   // UNICODE_TO_GBK[22326] := 16#76CE;
   // UNICODE_TO_GBK[22327] := 16#B0BB;
   // UNICODE_TO_GBK[22328] := 16#76CF;
   // UNICODE_TO_GBK[22329] := 16#D5B5;
   // UNICODE_TO_GBK[22330] := 16#76D0;
   // UNICODE_TO_GBK[22331] := 16#D1CE;
   // UNICODE_TO_GBK[22332] := 16#76D1;
   // UNICODE_TO_GBK[22333] := 16#BCE0;
   // UNICODE_TO_GBK[22334] := 16#76D2;
   // UNICODE_TO_GBK[22335] := 16#BAD0;
   // UNICODE_TO_GBK[22336] := 16#76D3;
   // UNICODE_TO_GBK[22337] := 16#B145;
   // UNICODE_TO_GBK[22338] := 16#76D4;
   // UNICODE_TO_GBK[22339] := 16#BFF8;
   // UNICODE_TO_GBK[22340] := 16#76D5;
   // UNICODE_TO_GBK[22341] := 16#B146;
   // UNICODE_TO_GBK[22342] := 16#76D6;
   // UNICODE_TO_GBK[22343] := 16#B8C7;
   // UNICODE_TO_GBK[22344] := 16#76D7;
   // UNICODE_TO_GBK[22345] := 16#B5C1;
   // UNICODE_TO_GBK[22346] := 16#76D8;
   // UNICODE_TO_GBK[22347] := 16#C5CC;
   // UNICODE_TO_GBK[22348] := 16#76D9;
   // UNICODE_TO_GBK[22349] := 16#B147;
   // UNICODE_TO_GBK[22350] := 16#76DA;
   // UNICODE_TO_GBK[22351] := 16#B148;
   // UNICODE_TO_GBK[22352] := 16#76DB;
   // UNICODE_TO_GBK[22353] := 16#CAA2;
   // UNICODE_TO_GBK[22354] := 16#76DC;
   // UNICODE_TO_GBK[22355] := 16#B149;
   // UNICODE_TO_GBK[22356] := 16#76DD;
   // UNICODE_TO_GBK[22357] := 16#B14A;
   // UNICODE_TO_GBK[22358] := 16#76DE;
   // UNICODE_TO_GBK[22359] := 16#B14B;
   // UNICODE_TO_GBK[22360] := 16#76DF;
   // UNICODE_TO_GBK[22361] := 16#C3CB;
   // UNICODE_TO_GBK[22362] := 16#76E0;
   // UNICODE_TO_GBK[22363] := 16#B14C;
   // UNICODE_TO_GBK[22364] := 16#76E1;
   // UNICODE_TO_GBK[22365] := 16#B14D;
   // UNICODE_TO_GBK[22366] := 16#76E2;
   // UNICODE_TO_GBK[22367] := 16#B14E;
   // UNICODE_TO_GBK[22368] := 16#76E3;
   // UNICODE_TO_GBK[22369] := 16#B14F;
   // UNICODE_TO_GBK[22370] := 16#76E4;
   // UNICODE_TO_GBK[22371] := 16#B150;
   // UNICODE_TO_GBK[22372] := 16#76E5;
   // UNICODE_TO_GBK[22373] := 16#EEC2;
   // UNICODE_TO_GBK[22374] := 16#76E6;
   // UNICODE_TO_GBK[22375] := 16#B151;
   // UNICODE_TO_GBK[22376] := 16#76E7;
   // UNICODE_TO_GBK[22377] := 16#B152;
   // UNICODE_TO_GBK[22378] := 16#76E8;
   // UNICODE_TO_GBK[22379] := 16#B153;
   // UNICODE_TO_GBK[22380] := 16#76E9;
   // UNICODE_TO_GBK[22381] := 16#B154;
   // UNICODE_TO_GBK[22382] := 16#76EA;
   // UNICODE_TO_GBK[22383] := 16#B155;
   // UNICODE_TO_GBK[22384] := 16#76EB;
   // UNICODE_TO_GBK[22385] := 16#B156;
   // UNICODE_TO_GBK[22386] := 16#76EC;
   // UNICODE_TO_GBK[22387] := 16#B157;
   // UNICODE_TO_GBK[22388] := 16#76ED;
   // UNICODE_TO_GBK[22389] := 16#B158;
   // UNICODE_TO_GBK[22390] := 16#76EE;
   // UNICODE_TO_GBK[22391] := 16#C4BF;
   // UNICODE_TO_GBK[22392] := 16#76EF;
   // UNICODE_TO_GBK[22393] := 16#B6A2;
   // UNICODE_TO_GBK[22394] := 16#76F0;
   // UNICODE_TO_GBK[22395] := 16#B159;
   // UNICODE_TO_GBK[22396] := 16#76F1;
   // UNICODE_TO_GBK[22397] := 16#EDEC;
   // UNICODE_TO_GBK[22398] := 16#76F2;
   // UNICODE_TO_GBK[22399] := 16#C3A4;
   // UNICODE_TO_GBK[22400] := 16#76F3;
   // UNICODE_TO_GBK[22401] := 16#B15A;
   // UNICODE_TO_GBK[22402] := 16#76F4;
   // UNICODE_TO_GBK[22403] := 16#D6B1;
   // UNICODE_TO_GBK[22404] := 16#76F5;
   // UNICODE_TO_GBK[22405] := 16#B15B;
   // UNICODE_TO_GBK[22406] := 16#76F6;
   // UNICODE_TO_GBK[22407] := 16#B15C;
   // UNICODE_TO_GBK[22408] := 16#76F7;
   // UNICODE_TO_GBK[22409] := 16#B15D;
   // UNICODE_TO_GBK[22410] := 16#76F8;
   // UNICODE_TO_GBK[22411] := 16#CFE0;
   // UNICODE_TO_GBK[22412] := 16#76F9;
   // UNICODE_TO_GBK[22413] := 16#EDEF;
   // UNICODE_TO_GBK[22414] := 16#76FA;
   // UNICODE_TO_GBK[22415] := 16#B15E;
   // UNICODE_TO_GBK[22416] := 16#76FB;
   // UNICODE_TO_GBK[22417] := 16#B15F;
   // UNICODE_TO_GBK[22418] := 16#76FC;
   // UNICODE_TO_GBK[22419] := 16#C5CE;
   // UNICODE_TO_GBK[22420] := 16#76FD;
   // UNICODE_TO_GBK[22421] := 16#B160;
   // UNICODE_TO_GBK[22422] := 16#76FE;
   // UNICODE_TO_GBK[22423] := 16#B6DC;
   // UNICODE_TO_GBK[22424] := 16#76FF;
   // UNICODE_TO_GBK[22425] := 16#B161;
   // UNICODE_TO_GBK[22426] := 16#7700;
   // UNICODE_TO_GBK[22427] := 16#B162;
   // UNICODE_TO_GBK[22428] := 16#7701;
   // UNICODE_TO_GBK[22429] := 16#CAA1;
   // UNICODE_TO_GBK[22430] := 16#7702;
   // UNICODE_TO_GBK[22431] := 16#B163;
   // UNICODE_TO_GBK[22432] := 16#7703;
   // UNICODE_TO_GBK[22433] := 16#B164;
   // UNICODE_TO_GBK[22434] := 16#7704;
   // UNICODE_TO_GBK[22435] := 16#EDED;
   // UNICODE_TO_GBK[22436] := 16#7705;
   // UNICODE_TO_GBK[22437] := 16#B165;
   // UNICODE_TO_GBK[22438] := 16#7706;
   // UNICODE_TO_GBK[22439] := 16#B166;
   // UNICODE_TO_GBK[22440] := 16#7707;
   // UNICODE_TO_GBK[22441] := 16#EDF0;
   // UNICODE_TO_GBK[22442] := 16#7708;
   // UNICODE_TO_GBK[22443] := 16#EDF1;
   // UNICODE_TO_GBK[22444] := 16#7709;
   // UNICODE_TO_GBK[22445] := 16#C3BC;
   // UNICODE_TO_GBK[22446] := 16#770A;
   // UNICODE_TO_GBK[22447] := 16#B167;
   // UNICODE_TO_GBK[22448] := 16#770B;
   // UNICODE_TO_GBK[22449] := 16#BFB4;
   // UNICODE_TO_GBK[22450] := 16#770C;
   // UNICODE_TO_GBK[22451] := 16#B168;
   // UNICODE_TO_GBK[22452] := 16#770D;
   // UNICODE_TO_GBK[22453] := 16#EDEE;
   // UNICODE_TO_GBK[22454] := 16#770E;
   // UNICODE_TO_GBK[22455] := 16#B169;
   // UNICODE_TO_GBK[22456] := 16#770F;
   // UNICODE_TO_GBK[22457] := 16#B16A;
   // UNICODE_TO_GBK[22458] := 16#7710;
   // UNICODE_TO_GBK[22459] := 16#B16B;
   // UNICODE_TO_GBK[22460] := 16#7711;
   // UNICODE_TO_GBK[22461] := 16#B16C;
   // UNICODE_TO_GBK[22462] := 16#7712;
   // UNICODE_TO_GBK[22463] := 16#B16D;
   // UNICODE_TO_GBK[22464] := 16#7713;
   // UNICODE_TO_GBK[22465] := 16#B16E;
   // UNICODE_TO_GBK[22466] := 16#7714;
   // UNICODE_TO_GBK[22467] := 16#B16F;
   // UNICODE_TO_GBK[22468] := 16#7715;
   // UNICODE_TO_GBK[22469] := 16#B170;
   // UNICODE_TO_GBK[22470] := 16#7716;
   // UNICODE_TO_GBK[22471] := 16#B171;
   // UNICODE_TO_GBK[22472] := 16#7717;
   // UNICODE_TO_GBK[22473] := 16#B172;
   // UNICODE_TO_GBK[22474] := 16#7718;
   // UNICODE_TO_GBK[22475] := 16#B173;
   // UNICODE_TO_GBK[22476] := 16#7719;
   // UNICODE_TO_GBK[22477] := 16#EDF4;
   // UNICODE_TO_GBK[22478] := 16#771A;
   // UNICODE_TO_GBK[22479] := 16#EDF2;
   // UNICODE_TO_GBK[22480] := 16#771B;
   // UNICODE_TO_GBK[22481] := 16#B174;
   // UNICODE_TO_GBK[22482] := 16#771C;
   // UNICODE_TO_GBK[22483] := 16#B175;
   // UNICODE_TO_GBK[22484] := 16#771D;
   // UNICODE_TO_GBK[22485] := 16#B176;
   // UNICODE_TO_GBK[22486] := 16#771E;
   // UNICODE_TO_GBK[22487] := 16#B177;
   // UNICODE_TO_GBK[22488] := 16#771F;
   // UNICODE_TO_GBK[22489] := 16#D5E6;
   // UNICODE_TO_GBK[22490] := 16#7720;
   // UNICODE_TO_GBK[22491] := 16#C3DF;
   // UNICODE_TO_GBK[22492] := 16#7721;
   // UNICODE_TO_GBK[22493] := 16#B178;
   // UNICODE_TO_GBK[22494] := 16#7722;
   // UNICODE_TO_GBK[22495] := 16#EDF3;
   // UNICODE_TO_GBK[22496] := 16#7723;
   // UNICODE_TO_GBK[22497] := 16#B179;
   // UNICODE_TO_GBK[22498] := 16#7724;
   // UNICODE_TO_GBK[22499] := 16#B17A;
   // UNICODE_TO_GBK[22500] := 16#7725;
   // UNICODE_TO_GBK[22501] := 16#B17B;
   // UNICODE_TO_GBK[22502] := 16#7726;
   // UNICODE_TO_GBK[22503] := 16#EDF6;
   // UNICODE_TO_GBK[22504] := 16#7727;
   // UNICODE_TO_GBK[22505] := 16#B17C;
   // UNICODE_TO_GBK[22506] := 16#7728;
   // UNICODE_TO_GBK[22507] := 16#D5A3;
   // UNICODE_TO_GBK[22508] := 16#7729;
   // UNICODE_TO_GBK[22509] := 16#D1A3;
   // UNICODE_TO_GBK[22510] := 16#772A;
   // UNICODE_TO_GBK[22511] := 16#B17D;
   // UNICODE_TO_GBK[22512] := 16#772B;
   // UNICODE_TO_GBK[22513] := 16#B17E;
   // UNICODE_TO_GBK[22514] := 16#772C;
   // UNICODE_TO_GBK[22515] := 16#B180;
   // UNICODE_TO_GBK[22516] := 16#772D;
   // UNICODE_TO_GBK[22517] := 16#EDF5;
   // UNICODE_TO_GBK[22518] := 16#772E;
   // UNICODE_TO_GBK[22519] := 16#B181;
   // UNICODE_TO_GBK[22520] := 16#772F;
   // UNICODE_TO_GBK[22521] := 16#C3D0;
   // UNICODE_TO_GBK[22522] := 16#7730;
   // UNICODE_TO_GBK[22523] := 16#B182;
   // UNICODE_TO_GBK[22524] := 16#7731;
   // UNICODE_TO_GBK[22525] := 16#B183;
   // UNICODE_TO_GBK[22526] := 16#7732;
   // UNICODE_TO_GBK[22527] := 16#B184;
   // UNICODE_TO_GBK[22528] := 16#7733;
   // UNICODE_TO_GBK[22529] := 16#B185;
   // UNICODE_TO_GBK[22530] := 16#7734;
   // UNICODE_TO_GBK[22531] := 16#B186;
   // UNICODE_TO_GBK[22532] := 16#7735;
   // UNICODE_TO_GBK[22533] := 16#EDF7;
   // UNICODE_TO_GBK[22534] := 16#7736;
   // UNICODE_TO_GBK[22535] := 16#BFF4;
   // UNICODE_TO_GBK[22536] := 16#7737;
   // UNICODE_TO_GBK[22537] := 16#BEEC;
   // UNICODE_TO_GBK[22538] := 16#7738;
   // UNICODE_TO_GBK[22539] := 16#EDF8;
   // UNICODE_TO_GBK[22540] := 16#7739;
   // UNICODE_TO_GBK[22541] := 16#B187;
   // UNICODE_TO_GBK[22542] := 16#773A;
   // UNICODE_TO_GBK[22543] := 16#CCF7;
   // UNICODE_TO_GBK[22544] := 16#773B;
   // UNICODE_TO_GBK[22545] := 16#B188;
   // UNICODE_TO_GBK[22546] := 16#773C;
   // UNICODE_TO_GBK[22547] := 16#D1DB;
   // UNICODE_TO_GBK[22548] := 16#773D;
   // UNICODE_TO_GBK[22549] := 16#B189;
   // UNICODE_TO_GBK[22550] := 16#773E;
   // UNICODE_TO_GBK[22551] := 16#B18A;
   // UNICODE_TO_GBK[22552] := 16#773F;
   // UNICODE_TO_GBK[22553] := 16#B18B;
   // UNICODE_TO_GBK[22554] := 16#7740;
   // UNICODE_TO_GBK[22555] := 16#D7C5;
   // UNICODE_TO_GBK[22556] := 16#7741;
   // UNICODE_TO_GBK[22557] := 16#D5F6;
   // UNICODE_TO_GBK[22558] := 16#7742;
   // UNICODE_TO_GBK[22559] := 16#B18C;
   // UNICODE_TO_GBK[22560] := 16#7743;
   // UNICODE_TO_GBK[22561] := 16#EDFC;
   // UNICODE_TO_GBK[22562] := 16#7744;
   // UNICODE_TO_GBK[22563] := 16#B18D;
   // UNICODE_TO_GBK[22564] := 16#7745;
   // UNICODE_TO_GBK[22565] := 16#B18E;
   // UNICODE_TO_GBK[22566] := 16#7746;
   // UNICODE_TO_GBK[22567] := 16#B18F;
   // UNICODE_TO_GBK[22568] := 16#7747;
   // UNICODE_TO_GBK[22569] := 16#EDFB;
   // UNICODE_TO_GBK[22570] := 16#7748;
   // UNICODE_TO_GBK[22571] := 16#B190;
   // UNICODE_TO_GBK[22572] := 16#7749;
   // UNICODE_TO_GBK[22573] := 16#B191;
   // UNICODE_TO_GBK[22574] := 16#774A;
   // UNICODE_TO_GBK[22575] := 16#B192;
   // UNICODE_TO_GBK[22576] := 16#774B;
   // UNICODE_TO_GBK[22577] := 16#B193;
   // UNICODE_TO_GBK[22578] := 16#774C;
   // UNICODE_TO_GBK[22579] := 16#B194;
   // UNICODE_TO_GBK[22580] := 16#774D;
   // UNICODE_TO_GBK[22581] := 16#B195;
   // UNICODE_TO_GBK[22582] := 16#774E;
   // UNICODE_TO_GBK[22583] := 16#B196;
   // UNICODE_TO_GBK[22584] := 16#774F;
   // UNICODE_TO_GBK[22585] := 16#B197;
   // UNICODE_TO_GBK[22586] := 16#7750;
   // UNICODE_TO_GBK[22587] := 16#EDF9;
   // UNICODE_TO_GBK[22588] := 16#7751;
   // UNICODE_TO_GBK[22589] := 16#EDFA;
   // UNICODE_TO_GBK[22590] := 16#7752;
   // UNICODE_TO_GBK[22591] := 16#B198;
   // UNICODE_TO_GBK[22592] := 16#7753;
   // UNICODE_TO_GBK[22593] := 16#B199;
   // UNICODE_TO_GBK[22594] := 16#7754;
   // UNICODE_TO_GBK[22595] := 16#B19A;
   // UNICODE_TO_GBK[22596] := 16#7755;
   // UNICODE_TO_GBK[22597] := 16#B19B;
   // UNICODE_TO_GBK[22598] := 16#7756;
   // UNICODE_TO_GBK[22599] := 16#B19C;
   // UNICODE_TO_GBK[22600] := 16#7757;
   // UNICODE_TO_GBK[22601] := 16#B19D;
   // UNICODE_TO_GBK[22602] := 16#7758;
   // UNICODE_TO_GBK[22603] := 16#B19E;
   // UNICODE_TO_GBK[22604] := 16#7759;
   // UNICODE_TO_GBK[22605] := 16#B19F;
   // UNICODE_TO_GBK[22606] := 16#775A;
   // UNICODE_TO_GBK[22607] := 16#EDFD;
   // UNICODE_TO_GBK[22608] := 16#775B;
   // UNICODE_TO_GBK[22609] := 16#BEA6;
   // UNICODE_TO_GBK[22610] := 16#775C;
   // UNICODE_TO_GBK[22611] := 16#B1A0;
   // UNICODE_TO_GBK[22612] := 16#775D;
   // UNICODE_TO_GBK[22613] := 16#B240;
   // UNICODE_TO_GBK[22614] := 16#775E;
   // UNICODE_TO_GBK[22615] := 16#B241;
   // UNICODE_TO_GBK[22616] := 16#775F;
   // UNICODE_TO_GBK[22617] := 16#B242;
   // UNICODE_TO_GBK[22618] := 16#7760;
   // UNICODE_TO_GBK[22619] := 16#B243;
   // UNICODE_TO_GBK[22620] := 16#7761;
   // UNICODE_TO_GBK[22621] := 16#CBAF;
   // UNICODE_TO_GBK[22622] := 16#7762;
   // UNICODE_TO_GBK[22623] := 16#EEA1;
   // UNICODE_TO_GBK[22624] := 16#7763;
   // UNICODE_TO_GBK[22625] := 16#B6BD;
   // UNICODE_TO_GBK[22626] := 16#7764;
   // UNICODE_TO_GBK[22627] := 16#B244;
   // UNICODE_TO_GBK[22628] := 16#7765;
   // UNICODE_TO_GBK[22629] := 16#EEA2;
   // UNICODE_TO_GBK[22630] := 16#7766;
   // UNICODE_TO_GBK[22631] := 16#C4C0;
   // UNICODE_TO_GBK[22632] := 16#7767;
   // UNICODE_TO_GBK[22633] := 16#B245;
   // UNICODE_TO_GBK[22634] := 16#7768;
   // UNICODE_TO_GBK[22635] := 16#EDFE;
   // UNICODE_TO_GBK[22636] := 16#7769;
   // UNICODE_TO_GBK[22637] := 16#B246;
   // UNICODE_TO_GBK[22638] := 16#776A;
   // UNICODE_TO_GBK[22639] := 16#B247;
   // UNICODE_TO_GBK[22640] := 16#776B;
   // UNICODE_TO_GBK[22641] := 16#BDDE;
   // UNICODE_TO_GBK[22642] := 16#776C;
   // UNICODE_TO_GBK[22643] := 16#B2C7;
   // UNICODE_TO_GBK[22644] := 16#776D;
   // UNICODE_TO_GBK[22645] := 16#B248;
   // UNICODE_TO_GBK[22646] := 16#776E;
   // UNICODE_TO_GBK[22647] := 16#B249;
   // UNICODE_TO_GBK[22648] := 16#776F;
   // UNICODE_TO_GBK[22649] := 16#B24A;
   // UNICODE_TO_GBK[22650] := 16#7770;
   // UNICODE_TO_GBK[22651] := 16#B24B;
   // UNICODE_TO_GBK[22652] := 16#7771;
   // UNICODE_TO_GBK[22653] := 16#B24C;
   // UNICODE_TO_GBK[22654] := 16#7772;
   // UNICODE_TO_GBK[22655] := 16#B24D;
   // UNICODE_TO_GBK[22656] := 16#7773;
   // UNICODE_TO_GBK[22657] := 16#B24E;
   // UNICODE_TO_GBK[22658] := 16#7774;
   // UNICODE_TO_GBK[22659] := 16#B24F;
   // UNICODE_TO_GBK[22660] := 16#7775;
   // UNICODE_TO_GBK[22661] := 16#B250;
   // UNICODE_TO_GBK[22662] := 16#7776;
   // UNICODE_TO_GBK[22663] := 16#B251;
   // UNICODE_TO_GBK[22664] := 16#7777;
   // UNICODE_TO_GBK[22665] := 16#B252;
   // UNICODE_TO_GBK[22666] := 16#7778;
   // UNICODE_TO_GBK[22667] := 16#B253;
   // UNICODE_TO_GBK[22668] := 16#7779;
   // UNICODE_TO_GBK[22669] := 16#B6C3;
   // UNICODE_TO_GBK[22670] := 16#777A;
   // UNICODE_TO_GBK[22671] := 16#B254;
   // UNICODE_TO_GBK[22672] := 16#777B;
   // UNICODE_TO_GBK[22673] := 16#B255;
   // UNICODE_TO_GBK[22674] := 16#777C;
   // UNICODE_TO_GBK[22675] := 16#B256;
   // UNICODE_TO_GBK[22676] := 16#777D;
   // UNICODE_TO_GBK[22677] := 16#EEA5;
   // UNICODE_TO_GBK[22678] := 16#777E;
   // UNICODE_TO_GBK[22679] := 16#D8BA;
   // UNICODE_TO_GBK[22680] := 16#777F;
   // UNICODE_TO_GBK[22681] := 16#EEA3;
   // UNICODE_TO_GBK[22682] := 16#7780;
   // UNICODE_TO_GBK[22683] := 16#EEA6;
   // UNICODE_TO_GBK[22684] := 16#7781;
   // UNICODE_TO_GBK[22685] := 16#B257;
   // UNICODE_TO_GBK[22686] := 16#7782;
   // UNICODE_TO_GBK[22687] := 16#B258;
   // UNICODE_TO_GBK[22688] := 16#7783;
   // UNICODE_TO_GBK[22689] := 16#B259;
   // UNICODE_TO_GBK[22690] := 16#7784;
   // UNICODE_TO_GBK[22691] := 16#C3E9;
   // UNICODE_TO_GBK[22692] := 16#7785;
   // UNICODE_TO_GBK[22693] := 16#B3F2;
   // UNICODE_TO_GBK[22694] := 16#7786;
   // UNICODE_TO_GBK[22695] := 16#B25A;
   // UNICODE_TO_GBK[22696] := 16#7787;
   // UNICODE_TO_GBK[22697] := 16#B25B;
   // UNICODE_TO_GBK[22698] := 16#7788;
   // UNICODE_TO_GBK[22699] := 16#B25C;
   // UNICODE_TO_GBK[22700] := 16#7789;
   // UNICODE_TO_GBK[22701] := 16#B25D;
   // UNICODE_TO_GBK[22702] := 16#778A;
   // UNICODE_TO_GBK[22703] := 16#B25E;
   // UNICODE_TO_GBK[22704] := 16#778B;
   // UNICODE_TO_GBK[22705] := 16#B25F;
   // UNICODE_TO_GBK[22706] := 16#778C;
   // UNICODE_TO_GBK[22707] := 16#EEA7;
   // UNICODE_TO_GBK[22708] := 16#778D;
   // UNICODE_TO_GBK[22709] := 16#EEA4;
   // UNICODE_TO_GBK[22710] := 16#778E;
   // UNICODE_TO_GBK[22711] := 16#CFB9;
   // UNICODE_TO_GBK[22712] := 16#778F;
   // UNICODE_TO_GBK[22713] := 16#B260;
   // UNICODE_TO_GBK[22714] := 16#7790;
   // UNICODE_TO_GBK[22715] := 16#B261;
   // UNICODE_TO_GBK[22716] := 16#7791;
   // UNICODE_TO_GBK[22717] := 16#EEA8;
   // UNICODE_TO_GBK[22718] := 16#7792;
   // UNICODE_TO_GBK[22719] := 16#C2F7;
   // UNICODE_TO_GBK[22720] := 16#7793;
   // UNICODE_TO_GBK[22721] := 16#B262;
   // UNICODE_TO_GBK[22722] := 16#7794;
   // UNICODE_TO_GBK[22723] := 16#B263;
   // UNICODE_TO_GBK[22724] := 16#7795;
   // UNICODE_TO_GBK[22725] := 16#B264;
   // UNICODE_TO_GBK[22726] := 16#7796;
   // UNICODE_TO_GBK[22727] := 16#B265;
   // UNICODE_TO_GBK[22728] := 16#7797;
   // UNICODE_TO_GBK[22729] := 16#B266;
   // UNICODE_TO_GBK[22730] := 16#7798;
   // UNICODE_TO_GBK[22731] := 16#B267;
   // UNICODE_TO_GBK[22732] := 16#7799;
   // UNICODE_TO_GBK[22733] := 16#B268;
   // UNICODE_TO_GBK[22734] := 16#779A;
   // UNICODE_TO_GBK[22735] := 16#B269;
   // UNICODE_TO_GBK[22736] := 16#779B;
   // UNICODE_TO_GBK[22737] := 16#B26A;
   // UNICODE_TO_GBK[22738] := 16#779C;
   // UNICODE_TO_GBK[22739] := 16#B26B;
   // UNICODE_TO_GBK[22740] := 16#779D;
   // UNICODE_TO_GBK[22741] := 16#B26C;
   // UNICODE_TO_GBK[22742] := 16#779E;
   // UNICODE_TO_GBK[22743] := 16#B26D;
   // UNICODE_TO_GBK[22744] := 16#779F;
   // UNICODE_TO_GBK[22745] := 16#EEA9;
   // UNICODE_TO_GBK[22746] := 16#77A0;
   // UNICODE_TO_GBK[22747] := 16#EEAA;
   // UNICODE_TO_GBK[22748] := 16#77A1;
   // UNICODE_TO_GBK[22749] := 16#B26E;
   // UNICODE_TO_GBK[22750] := 16#77A2;
   // UNICODE_TO_GBK[22751] := 16#DEAB;
   // UNICODE_TO_GBK[22752] := 16#77A3;
   // UNICODE_TO_GBK[22753] := 16#B26F;
   // UNICODE_TO_GBK[22754] := 16#77A4;
   // UNICODE_TO_GBK[22755] := 16#B270;
   // UNICODE_TO_GBK[22756] := 16#77A5;
   // UNICODE_TO_GBK[22757] := 16#C6B3;
   // UNICODE_TO_GBK[22758] := 16#77A6;
   // UNICODE_TO_GBK[22759] := 16#B271;
   // UNICODE_TO_GBK[22760] := 16#77A7;
   // UNICODE_TO_GBK[22761] := 16#C7C6;
   // UNICODE_TO_GBK[22762] := 16#77A8;
   // UNICODE_TO_GBK[22763] := 16#B272;
   // UNICODE_TO_GBK[22764] := 16#77A9;
   // UNICODE_TO_GBK[22765] := 16#D6F5;
   // UNICODE_TO_GBK[22766] := 16#77AA;
   // UNICODE_TO_GBK[22767] := 16#B5C9;
   // UNICODE_TO_GBK[22768] := 16#77AB;
   // UNICODE_TO_GBK[22769] := 16#B273;
   // UNICODE_TO_GBK[22770] := 16#77AC;
   // UNICODE_TO_GBK[22771] := 16#CBB2;
   // UNICODE_TO_GBK[22772] := 16#77AD;
   // UNICODE_TO_GBK[22773] := 16#B274;
   // UNICODE_TO_GBK[22774] := 16#77AE;
   // UNICODE_TO_GBK[22775] := 16#B275;
   // UNICODE_TO_GBK[22776] := 16#77AF;
   // UNICODE_TO_GBK[22777] := 16#B276;
   // UNICODE_TO_GBK[22778] := 16#77B0;
   // UNICODE_TO_GBK[22779] := 16#EEAB;
   // UNICODE_TO_GBK[22780] := 16#77B1;
   // UNICODE_TO_GBK[22781] := 16#B277;
   // UNICODE_TO_GBK[22782] := 16#77B2;
   // UNICODE_TO_GBK[22783] := 16#B278;
   // UNICODE_TO_GBK[22784] := 16#77B3;
   // UNICODE_TO_GBK[22785] := 16#CDAB;
   // UNICODE_TO_GBK[22786] := 16#77B4;
   // UNICODE_TO_GBK[22787] := 16#B279;
   // UNICODE_TO_GBK[22788] := 16#77B5;
   // UNICODE_TO_GBK[22789] := 16#EEAC;
   // UNICODE_TO_GBK[22790] := 16#77B6;
   // UNICODE_TO_GBK[22791] := 16#B27A;
   // UNICODE_TO_GBK[22792] := 16#77B7;
   // UNICODE_TO_GBK[22793] := 16#B27B;
   // UNICODE_TO_GBK[22794] := 16#77B8;
   // UNICODE_TO_GBK[22795] := 16#B27C;
   // UNICODE_TO_GBK[22796] := 16#77B9;
   // UNICODE_TO_GBK[22797] := 16#B27D;
   // UNICODE_TO_GBK[22798] := 16#77BA;
   // UNICODE_TO_GBK[22799] := 16#B27E;
   // UNICODE_TO_GBK[22800] := 16#77BB;
   // UNICODE_TO_GBK[22801] := 16#D5B0;
   // UNICODE_TO_GBK[22802] := 16#77BC;
   // UNICODE_TO_GBK[22803] := 16#B280;
   // UNICODE_TO_GBK[22804] := 16#77BD;
   // UNICODE_TO_GBK[22805] := 16#EEAD;
   // UNICODE_TO_GBK[22806] := 16#77BE;
   // UNICODE_TO_GBK[22807] := 16#B281;
   // UNICODE_TO_GBK[22808] := 16#77BF;
   // UNICODE_TO_GBK[22809] := 16#F6C4;
   // UNICODE_TO_GBK[22810] := 16#77C0;
   // UNICODE_TO_GBK[22811] := 16#B282;
   // UNICODE_TO_GBK[22812] := 16#77C1;
   // UNICODE_TO_GBK[22813] := 16#B283;
   // UNICODE_TO_GBK[22814] := 16#77C2;
   // UNICODE_TO_GBK[22815] := 16#B284;
   // UNICODE_TO_GBK[22816] := 16#77C3;
   // UNICODE_TO_GBK[22817] := 16#B285;
   // UNICODE_TO_GBK[22818] := 16#77C4;
   // UNICODE_TO_GBK[22819] := 16#B286;
   // UNICODE_TO_GBK[22820] := 16#77C5;
   // UNICODE_TO_GBK[22821] := 16#B287;
   // UNICODE_TO_GBK[22822] := 16#77C6;
   // UNICODE_TO_GBK[22823] := 16#B288;
   // UNICODE_TO_GBK[22824] := 16#77C7;
   // UNICODE_TO_GBK[22825] := 16#B289;
   // UNICODE_TO_GBK[22826] := 16#77C8;
   // UNICODE_TO_GBK[22827] := 16#B28A;
   // UNICODE_TO_GBK[22828] := 16#77C9;
   // UNICODE_TO_GBK[22829] := 16#B28B;
   // UNICODE_TO_GBK[22830] := 16#77CA;
   // UNICODE_TO_GBK[22831] := 16#B28C;
   // UNICODE_TO_GBK[22832] := 16#77CB;
   // UNICODE_TO_GBK[22833] := 16#B28D;
   // UNICODE_TO_GBK[22834] := 16#77CC;
   // UNICODE_TO_GBK[22835] := 16#B28E;
   // UNICODE_TO_GBK[22836] := 16#77CD;
   // UNICODE_TO_GBK[22837] := 16#DBC7;
   // UNICODE_TO_GBK[22838] := 16#77CE;
   // UNICODE_TO_GBK[22839] := 16#B28F;
   // UNICODE_TO_GBK[22840] := 16#77CF;
   // UNICODE_TO_GBK[22841] := 16#B290;
   // UNICODE_TO_GBK[22842] := 16#77D0;
   // UNICODE_TO_GBK[22843] := 16#B291;
   // UNICODE_TO_GBK[22844] := 16#77D1;
   // UNICODE_TO_GBK[22845] := 16#B292;
   // UNICODE_TO_GBK[22846] := 16#77D2;
   // UNICODE_TO_GBK[22847] := 16#B293;
   // UNICODE_TO_GBK[22848] := 16#77D3;
   // UNICODE_TO_GBK[22849] := 16#B294;
   // UNICODE_TO_GBK[22850] := 16#77D4;
   // UNICODE_TO_GBK[22851] := 16#B295;
   // UNICODE_TO_GBK[22852] := 16#77D5;
   // UNICODE_TO_GBK[22853] := 16#B296;
   // UNICODE_TO_GBK[22854] := 16#77D6;
   // UNICODE_TO_GBK[22855] := 16#B297;
   // UNICODE_TO_GBK[22856] := 16#77D7;
   // UNICODE_TO_GBK[22857] := 16#B4A3;
   // UNICODE_TO_GBK[22858] := 16#77D8;
   // UNICODE_TO_GBK[22859] := 16#B298;
   // UNICODE_TO_GBK[22860] := 16#77D9;
   // UNICODE_TO_GBK[22861] := 16#B299;
   // UNICODE_TO_GBK[22862] := 16#77DA;
   // UNICODE_TO_GBK[22863] := 16#B29A;
   // UNICODE_TO_GBK[22864] := 16#77DB;
   // UNICODE_TO_GBK[22865] := 16#C3AC;
   // UNICODE_TO_GBK[22866] := 16#77DC;
   // UNICODE_TO_GBK[22867] := 16#F1E6;
   // UNICODE_TO_GBK[22868] := 16#77DD;
   // UNICODE_TO_GBK[22869] := 16#B29B;
   // UNICODE_TO_GBK[22870] := 16#77DE;
   // UNICODE_TO_GBK[22871] := 16#B29C;
   // UNICODE_TO_GBK[22872] := 16#77DF;
   // UNICODE_TO_GBK[22873] := 16#B29D;
   // UNICODE_TO_GBK[22874] := 16#77E0;
   // UNICODE_TO_GBK[22875] := 16#B29E;
   // UNICODE_TO_GBK[22876] := 16#77E1;
   // UNICODE_TO_GBK[22877] := 16#B29F;
   // UNICODE_TO_GBK[22878] := 16#77E2;
   // UNICODE_TO_GBK[22879] := 16#CAB8;
   // UNICODE_TO_GBK[22880] := 16#77E3;
   // UNICODE_TO_GBK[22881] := 16#D2D3;
   // UNICODE_TO_GBK[22882] := 16#77E4;
   // UNICODE_TO_GBK[22883] := 16#B2A0;
   // UNICODE_TO_GBK[22884] := 16#77E5;
   // UNICODE_TO_GBK[22885] := 16#D6AA;
   // UNICODE_TO_GBK[22886] := 16#77E6;
   // UNICODE_TO_GBK[22887] := 16#B340;
   // UNICODE_TO_GBK[22888] := 16#77E7;
   // UNICODE_TO_GBK[22889] := 16#EFF2;
   // UNICODE_TO_GBK[22890] := 16#77E8;
   // UNICODE_TO_GBK[22891] := 16#B341;
   // UNICODE_TO_GBK[22892] := 16#77E9;
   // UNICODE_TO_GBK[22893] := 16#BED8;
   // UNICODE_TO_GBK[22894] := 16#77EA;
   // UNICODE_TO_GBK[22895] := 16#B342;
   // UNICODE_TO_GBK[22896] := 16#77EB;
   // UNICODE_TO_GBK[22897] := 16#BDC3;
   // UNICODE_TO_GBK[22898] := 16#77EC;
   // UNICODE_TO_GBK[22899] := 16#EFF3;
   // UNICODE_TO_GBK[22900] := 16#77ED;
   // UNICODE_TO_GBK[22901] := 16#B6CC;
   // UNICODE_TO_GBK[22902] := 16#77EE;
   // UNICODE_TO_GBK[22903] := 16#B0AB;
   // UNICODE_TO_GBK[22904] := 16#77EF;
   // UNICODE_TO_GBK[22905] := 16#B343;
   // UNICODE_TO_GBK[22906] := 16#77F0;
   // UNICODE_TO_GBK[22907] := 16#B344;
   // UNICODE_TO_GBK[22908] := 16#77F1;
   // UNICODE_TO_GBK[22909] := 16#B345;
   // UNICODE_TO_GBK[22910] := 16#77F2;
   // UNICODE_TO_GBK[22911] := 16#B346;
   // UNICODE_TO_GBK[22912] := 16#77F3;
   // UNICODE_TO_GBK[22913] := 16#CAAF;
   // UNICODE_TO_GBK[22914] := 16#77F4;
   // UNICODE_TO_GBK[22915] := 16#B347;
   // UNICODE_TO_GBK[22916] := 16#77F5;
   // UNICODE_TO_GBK[22917] := 16#B348;
   // UNICODE_TO_GBK[22918] := 16#77F6;
   // UNICODE_TO_GBK[22919] := 16#EDB6;
   // UNICODE_TO_GBK[22920] := 16#77F7;
   // UNICODE_TO_GBK[22921] := 16#B349;
   // UNICODE_TO_GBK[22922] := 16#77F8;
   // UNICODE_TO_GBK[22923] := 16#EDB7;
   // UNICODE_TO_GBK[22924] := 16#77F9;
   // UNICODE_TO_GBK[22925] := 16#B34A;
   // UNICODE_TO_GBK[22926] := 16#77FA;
   // UNICODE_TO_GBK[22927] := 16#B34B;
   // UNICODE_TO_GBK[22928] := 16#77FB;
   // UNICODE_TO_GBK[22929] := 16#B34C;
   // UNICODE_TO_GBK[22930] := 16#77FC;
   // UNICODE_TO_GBK[22931] := 16#B34D;
   // UNICODE_TO_GBK[22932] := 16#77FD;
   // UNICODE_TO_GBK[22933] := 16#CEF9;
   // UNICODE_TO_GBK[22934] := 16#77FE;
   // UNICODE_TO_GBK[22935] := 16#B7AF;
   // UNICODE_TO_GBK[22936] := 16#77FF;
   // UNICODE_TO_GBK[22937] := 16#BFF3;
   // UNICODE_TO_GBK[22938] := 16#7800;
   // UNICODE_TO_GBK[22939] := 16#EDB8;
   // UNICODE_TO_GBK[22940] := 16#7801;
   // UNICODE_TO_GBK[22941] := 16#C2EB;
   // UNICODE_TO_GBK[22942] := 16#7802;
   // UNICODE_TO_GBK[22943] := 16#C9B0;
   // UNICODE_TO_GBK[22944] := 16#7803;
   // UNICODE_TO_GBK[22945] := 16#B34E;
   // UNICODE_TO_GBK[22946] := 16#7804;
   // UNICODE_TO_GBK[22947] := 16#B34F;
   // UNICODE_TO_GBK[22948] := 16#7805;
   // UNICODE_TO_GBK[22949] := 16#B350;
   // UNICODE_TO_GBK[22950] := 16#7806;
   // UNICODE_TO_GBK[22951] := 16#B351;
   // UNICODE_TO_GBK[22952] := 16#7807;
   // UNICODE_TO_GBK[22953] := 16#B352;
   // UNICODE_TO_GBK[22954] := 16#7808;
   // UNICODE_TO_GBK[22955] := 16#B353;
   // UNICODE_TO_GBK[22956] := 16#7809;
   // UNICODE_TO_GBK[22957] := 16#EDB9;
   // UNICODE_TO_GBK[22958] := 16#780A;
   // UNICODE_TO_GBK[22959] := 16#B354;
   // UNICODE_TO_GBK[22960] := 16#780B;
   // UNICODE_TO_GBK[22961] := 16#B355;
   // UNICODE_TO_GBK[22962] := 16#780C;
   // UNICODE_TO_GBK[22963] := 16#C6F6;
   // UNICODE_TO_GBK[22964] := 16#780D;
   // UNICODE_TO_GBK[22965] := 16#BFB3;
   // UNICODE_TO_GBK[22966] := 16#780E;
   // UNICODE_TO_GBK[22967] := 16#B356;
   // UNICODE_TO_GBK[22968] := 16#780F;
   // UNICODE_TO_GBK[22969] := 16#B357;
   // UNICODE_TO_GBK[22970] := 16#7810;
   // UNICODE_TO_GBK[22971] := 16#B358;
   // UNICODE_TO_GBK[22972] := 16#7811;
   // UNICODE_TO_GBK[22973] := 16#EDBC;
   // UNICODE_TO_GBK[22974] := 16#7812;
   // UNICODE_TO_GBK[22975] := 16#C5F8;
   // UNICODE_TO_GBK[22976] := 16#7813;
   // UNICODE_TO_GBK[22977] := 16#B359;
   // UNICODE_TO_GBK[22978] := 16#7814;
   // UNICODE_TO_GBK[22979] := 16#D1D0;
   // UNICODE_TO_GBK[22980] := 16#7815;
   // UNICODE_TO_GBK[22981] := 16#B35A;
   // UNICODE_TO_GBK[22982] := 16#7816;
   // UNICODE_TO_GBK[22983] := 16#D7A9;
   // UNICODE_TO_GBK[22984] := 16#7817;
   // UNICODE_TO_GBK[22985] := 16#EDBA;
   // UNICODE_TO_GBK[22986] := 16#7818;
   // UNICODE_TO_GBK[22987] := 16#EDBB;
   // UNICODE_TO_GBK[22988] := 16#7819;
   // UNICODE_TO_GBK[22989] := 16#B35B;
   // UNICODE_TO_GBK[22990] := 16#781A;
   // UNICODE_TO_GBK[22991] := 16#D1E2;
   // UNICODE_TO_GBK[22992] := 16#781B;
   // UNICODE_TO_GBK[22993] := 16#B35C;
   // UNICODE_TO_GBK[22994] := 16#781C;
   // UNICODE_TO_GBK[22995] := 16#EDBF;
   // UNICODE_TO_GBK[22996] := 16#781D;
   // UNICODE_TO_GBK[22997] := 16#EDC0;
   // UNICODE_TO_GBK[22998] := 16#781E;
   // UNICODE_TO_GBK[22999] := 16#B35D;
   // UNICODE_TO_GBK[23000] := 16#781F;
   // UNICODE_TO_GBK[23001] := 16#EDC4;
   // UNICODE_TO_GBK[23002] := 16#7820;
   // UNICODE_TO_GBK[23003] := 16#B35E;
   // UNICODE_TO_GBK[23004] := 16#7821;
   // UNICODE_TO_GBK[23005] := 16#B35F;
   // UNICODE_TO_GBK[23006] := 16#7822;
   // UNICODE_TO_GBK[23007] := 16#B360;
   // UNICODE_TO_GBK[23008] := 16#7823;
   // UNICODE_TO_GBK[23009] := 16#EDC8;
   // UNICODE_TO_GBK[23010] := 16#7824;
   // UNICODE_TO_GBK[23011] := 16#B361;
   // UNICODE_TO_GBK[23012] := 16#7825;
   // UNICODE_TO_GBK[23013] := 16#EDC6;
   // UNICODE_TO_GBK[23014] := 16#7826;
   // UNICODE_TO_GBK[23015] := 16#EDCE;
   // UNICODE_TO_GBK[23016] := 16#7827;
   // UNICODE_TO_GBK[23017] := 16#D5E8;
   // UNICODE_TO_GBK[23018] := 16#7828;
   // UNICODE_TO_GBK[23019] := 16#B362;
   // UNICODE_TO_GBK[23020] := 16#7829;
   // UNICODE_TO_GBK[23021] := 16#EDC9;
   // UNICODE_TO_GBK[23022] := 16#782A;
   // UNICODE_TO_GBK[23023] := 16#B363;
   // UNICODE_TO_GBK[23024] := 16#782B;
   // UNICODE_TO_GBK[23025] := 16#B364;
   // UNICODE_TO_GBK[23026] := 16#782C;
   // UNICODE_TO_GBK[23027] := 16#EDC7;
   // UNICODE_TO_GBK[23028] := 16#782D;
   // UNICODE_TO_GBK[23029] := 16#EDBE;
   // UNICODE_TO_GBK[23030] := 16#782E;
   // UNICODE_TO_GBK[23031] := 16#B365;
   // UNICODE_TO_GBK[23032] := 16#782F;
   // UNICODE_TO_GBK[23033] := 16#B366;
   // UNICODE_TO_GBK[23034] := 16#7830;
   // UNICODE_TO_GBK[23035] := 16#C5E9;
   // UNICODE_TO_GBK[23036] := 16#7831;
   // UNICODE_TO_GBK[23037] := 16#B367;
   // UNICODE_TO_GBK[23038] := 16#7832;
   // UNICODE_TO_GBK[23039] := 16#B368;
   // UNICODE_TO_GBK[23040] := 16#7833;
   // UNICODE_TO_GBK[23041] := 16#B369;
   // UNICODE_TO_GBK[23042] := 16#7834;
   // UNICODE_TO_GBK[23043] := 16#C6C6;
   // UNICODE_TO_GBK[23044] := 16#7835;
   // UNICODE_TO_GBK[23045] := 16#B36A;
   // UNICODE_TO_GBK[23046] := 16#7836;
   // UNICODE_TO_GBK[23047] := 16#B36B;
   // UNICODE_TO_GBK[23048] := 16#7837;
   // UNICODE_TO_GBK[23049] := 16#C9E9;
   // UNICODE_TO_GBK[23050] := 16#7838;
   // UNICODE_TO_GBK[23051] := 16#D4D2;
   // UNICODE_TO_GBK[23052] := 16#7839;
   // UNICODE_TO_GBK[23053] := 16#EDC1;
   // UNICODE_TO_GBK[23054] := 16#783A;
   // UNICODE_TO_GBK[23055] := 16#EDC2;
   // UNICODE_TO_GBK[23056] := 16#783B;
   // UNICODE_TO_GBK[23057] := 16#EDC3;
   // UNICODE_TO_GBK[23058] := 16#783C;
   // UNICODE_TO_GBK[23059] := 16#EDC5;
   // UNICODE_TO_GBK[23060] := 16#783D;
   // UNICODE_TO_GBK[23061] := 16#B36C;
   // UNICODE_TO_GBK[23062] := 16#783E;
   // UNICODE_TO_GBK[23063] := 16#C0F9;
   // UNICODE_TO_GBK[23064] := 16#783F;
   // UNICODE_TO_GBK[23065] := 16#B36D;
   // UNICODE_TO_GBK[23066] := 16#7840;
   // UNICODE_TO_GBK[23067] := 16#B4A1;
   // UNICODE_TO_GBK[23068] := 16#7841;
   // UNICODE_TO_GBK[23069] := 16#B36E;
   // UNICODE_TO_GBK[23070] := 16#7842;
   // UNICODE_TO_GBK[23071] := 16#B36F;
   // UNICODE_TO_GBK[23072] := 16#7843;
   // UNICODE_TO_GBK[23073] := 16#B370;
   // UNICODE_TO_GBK[23074] := 16#7844;
   // UNICODE_TO_GBK[23075] := 16#B371;
   // UNICODE_TO_GBK[23076] := 16#7845;
   // UNICODE_TO_GBK[23077] := 16#B9E8;
   // UNICODE_TO_GBK[23078] := 16#7846;
   // UNICODE_TO_GBK[23079] := 16#B372;
   // UNICODE_TO_GBK[23080] := 16#7847;
   // UNICODE_TO_GBK[23081] := 16#EDD0;
   // UNICODE_TO_GBK[23082] := 16#7848;
   // UNICODE_TO_GBK[23083] := 16#B373;
   // UNICODE_TO_GBK[23084] := 16#7849;
   // UNICODE_TO_GBK[23085] := 16#B374;
   // UNICODE_TO_GBK[23086] := 16#784A;
   // UNICODE_TO_GBK[23087] := 16#B375;
   // UNICODE_TO_GBK[23088] := 16#784B;
   // UNICODE_TO_GBK[23089] := 16#B376;
   // UNICODE_TO_GBK[23090] := 16#784C;
   // UNICODE_TO_GBK[23091] := 16#EDD1;
   // UNICODE_TO_GBK[23092] := 16#784D;
   // UNICODE_TO_GBK[23093] := 16#B377;
   // UNICODE_TO_GBK[23094] := 16#784E;
   // UNICODE_TO_GBK[23095] := 16#EDCA;
   // UNICODE_TO_GBK[23096] := 16#784F;
   // UNICODE_TO_GBK[23097] := 16#B378;
   // UNICODE_TO_GBK[23098] := 16#7850;
   // UNICODE_TO_GBK[23099] := 16#EDCF;
   // UNICODE_TO_GBK[23100] := 16#7851;
   // UNICODE_TO_GBK[23101] := 16#B379;
   // UNICODE_TO_GBK[23102] := 16#7852;
   // UNICODE_TO_GBK[23103] := 16#CEF8;
   // UNICODE_TO_GBK[23104] := 16#7853;
   // UNICODE_TO_GBK[23105] := 16#B37A;
   // UNICODE_TO_GBK[23106] := 16#7854;
   // UNICODE_TO_GBK[23107] := 16#B37B;
   // UNICODE_TO_GBK[23108] := 16#7855;
   // UNICODE_TO_GBK[23109] := 16#CBB6;
   // UNICODE_TO_GBK[23110] := 16#7856;
   // UNICODE_TO_GBK[23111] := 16#EDCC;
   // UNICODE_TO_GBK[23112] := 16#7857;
   // UNICODE_TO_GBK[23113] := 16#EDCD;
   // UNICODE_TO_GBK[23114] := 16#7858;
   // UNICODE_TO_GBK[23115] := 16#B37C;
   // UNICODE_TO_GBK[23116] := 16#7859;
   // UNICODE_TO_GBK[23117] := 16#B37D;
   // UNICODE_TO_GBK[23118] := 16#785A;
   // UNICODE_TO_GBK[23119] := 16#B37E;
   // UNICODE_TO_GBK[23120] := 16#785B;
   // UNICODE_TO_GBK[23121] := 16#B380;
   // UNICODE_TO_GBK[23122] := 16#785C;
   // UNICODE_TO_GBK[23123] := 16#B381;
   // UNICODE_TO_GBK[23124] := 16#785D;
   // UNICODE_TO_GBK[23125] := 16#CFF5;
   // UNICODE_TO_GBK[23126] := 16#785E;
   // UNICODE_TO_GBK[23127] := 16#B382;
   // UNICODE_TO_GBK[23128] := 16#785F;
   // UNICODE_TO_GBK[23129] := 16#B383;
   // UNICODE_TO_GBK[23130] := 16#7860;
   // UNICODE_TO_GBK[23131] := 16#B384;
   // UNICODE_TO_GBK[23132] := 16#7861;
   // UNICODE_TO_GBK[23133] := 16#B385;
   // UNICODE_TO_GBK[23134] := 16#7862;
   // UNICODE_TO_GBK[23135] := 16#B386;
   // UNICODE_TO_GBK[23136] := 16#7863;
   // UNICODE_TO_GBK[23137] := 16#B387;
   // UNICODE_TO_GBK[23138] := 16#7864;
   // UNICODE_TO_GBK[23139] := 16#B388;
   // UNICODE_TO_GBK[23140] := 16#7865;
   // UNICODE_TO_GBK[23141] := 16#B389;
   // UNICODE_TO_GBK[23142] := 16#7866;
   // UNICODE_TO_GBK[23143] := 16#B38A;
   // UNICODE_TO_GBK[23144] := 16#7867;
   // UNICODE_TO_GBK[23145] := 16#B38B;
   // UNICODE_TO_GBK[23146] := 16#7868;
   // UNICODE_TO_GBK[23147] := 16#B38C;
   // UNICODE_TO_GBK[23148] := 16#7869;
   // UNICODE_TO_GBK[23149] := 16#B38D;
   // UNICODE_TO_GBK[23150] := 16#786A;
   // UNICODE_TO_GBK[23151] := 16#EDD2;
   // UNICODE_TO_GBK[23152] := 16#786B;
   // UNICODE_TO_GBK[23153] := 16#C1F2;
   // UNICODE_TO_GBK[23154] := 16#786C;
   // UNICODE_TO_GBK[23155] := 16#D3B2;
   // UNICODE_TO_GBK[23156] := 16#786D;
   // UNICODE_TO_GBK[23157] := 16#EDCB;
   // UNICODE_TO_GBK[23158] := 16#786E;
   // UNICODE_TO_GBK[23159] := 16#C8B7;
   // UNICODE_TO_GBK[23160] := 16#786F;
   // UNICODE_TO_GBK[23161] := 16#B38E;
   // UNICODE_TO_GBK[23162] := 16#7870;
   // UNICODE_TO_GBK[23163] := 16#B38F;
   // UNICODE_TO_GBK[23164] := 16#7871;
   // UNICODE_TO_GBK[23165] := 16#B390;
   // UNICODE_TO_GBK[23166] := 16#7872;
   // UNICODE_TO_GBK[23167] := 16#B391;
   // UNICODE_TO_GBK[23168] := 16#7873;
   // UNICODE_TO_GBK[23169] := 16#B392;
   // UNICODE_TO_GBK[23170] := 16#7874;
   // UNICODE_TO_GBK[23171] := 16#B393;
   // UNICODE_TO_GBK[23172] := 16#7875;
   // UNICODE_TO_GBK[23173] := 16#B394;
   // UNICODE_TO_GBK[23174] := 16#7876;
   // UNICODE_TO_GBK[23175] := 16#B395;
   // UNICODE_TO_GBK[23176] := 16#7877;
   // UNICODE_TO_GBK[23177] := 16#BCEF;
   // UNICODE_TO_GBK[23178] := 16#7878;
   // UNICODE_TO_GBK[23179] := 16#B396;
   // UNICODE_TO_GBK[23180] := 16#7879;
   // UNICODE_TO_GBK[23181] := 16#B397;
   // UNICODE_TO_GBK[23182] := 16#787A;
   // UNICODE_TO_GBK[23183] := 16#B398;
   // UNICODE_TO_GBK[23184] := 16#787B;
   // UNICODE_TO_GBK[23185] := 16#B399;
   // UNICODE_TO_GBK[23186] := 16#787C;
   // UNICODE_TO_GBK[23187] := 16#C5F0;
   // UNICODE_TO_GBK[23188] := 16#787D;
   // UNICODE_TO_GBK[23189] := 16#B39A;
   // UNICODE_TO_GBK[23190] := 16#787E;
   // UNICODE_TO_GBK[23191] := 16#B39B;
   // UNICODE_TO_GBK[23192] := 16#787F;
   // UNICODE_TO_GBK[23193] := 16#B39C;
   // UNICODE_TO_GBK[23194] := 16#7880;
   // UNICODE_TO_GBK[23195] := 16#B39D;
   // UNICODE_TO_GBK[23196] := 16#7881;
   // UNICODE_TO_GBK[23197] := 16#B39E;
   // UNICODE_TO_GBK[23198] := 16#7882;
   // UNICODE_TO_GBK[23199] := 16#B39F;
   // UNICODE_TO_GBK[23200] := 16#7883;
   // UNICODE_TO_GBK[23201] := 16#B3A0;
   // UNICODE_TO_GBK[23202] := 16#7884;
   // UNICODE_TO_GBK[23203] := 16#B440;
   // UNICODE_TO_GBK[23204] := 16#7885;
   // UNICODE_TO_GBK[23205] := 16#B441;
   // UNICODE_TO_GBK[23206] := 16#7886;
   // UNICODE_TO_GBK[23207] := 16#B442;
   // UNICODE_TO_GBK[23208] := 16#7887;
   // UNICODE_TO_GBK[23209] := 16#EDD6;
   // UNICODE_TO_GBK[23210] := 16#7888;
   // UNICODE_TO_GBK[23211] := 16#B443;
   // UNICODE_TO_GBK[23212] := 16#7889;
   // UNICODE_TO_GBK[23213] := 16#B5EF;
   // UNICODE_TO_GBK[23214] := 16#788A;
   // UNICODE_TO_GBK[23215] := 16#B444;
   // UNICODE_TO_GBK[23216] := 16#788B;
   // UNICODE_TO_GBK[23217] := 16#B445;
   // UNICODE_TO_GBK[23218] := 16#788C;
   // UNICODE_TO_GBK[23219] := 16#C2B5;
   // UNICODE_TO_GBK[23220] := 16#788D;
   // UNICODE_TO_GBK[23221] := 16#B0AD;
   // UNICODE_TO_GBK[23222] := 16#788E;
   // UNICODE_TO_GBK[23223] := 16#CBE9;
   // UNICODE_TO_GBK[23224] := 16#788F;
   // UNICODE_TO_GBK[23225] := 16#B446;
   // UNICODE_TO_GBK[23226] := 16#7890;
   // UNICODE_TO_GBK[23227] := 16#B447;
   // UNICODE_TO_GBK[23228] := 16#7891;
   // UNICODE_TO_GBK[23229] := 16#B1AE;
   // UNICODE_TO_GBK[23230] := 16#7892;
   // UNICODE_TO_GBK[23231] := 16#B448;
   // UNICODE_TO_GBK[23232] := 16#7893;
   // UNICODE_TO_GBK[23233] := 16#EDD4;
   // UNICODE_TO_GBK[23234] := 16#7894;
   // UNICODE_TO_GBK[23235] := 16#B449;
   // UNICODE_TO_GBK[23236] := 16#7895;
   // UNICODE_TO_GBK[23237] := 16#B44A;
   // UNICODE_TO_GBK[23238] := 16#7896;
   // UNICODE_TO_GBK[23239] := 16#B44B;
   // UNICODE_TO_GBK[23240] := 16#7897;
   // UNICODE_TO_GBK[23241] := 16#CDEB;
   // UNICODE_TO_GBK[23242] := 16#7898;
   // UNICODE_TO_GBK[23243] := 16#B5E2;
   // UNICODE_TO_GBK[23244] := 16#7899;
   // UNICODE_TO_GBK[23245] := 16#B44C;
   // UNICODE_TO_GBK[23246] := 16#789A;
   // UNICODE_TO_GBK[23247] := 16#EDD5;
   // UNICODE_TO_GBK[23248] := 16#789B;
   // UNICODE_TO_GBK[23249] := 16#EDD3;
   // UNICODE_TO_GBK[23250] := 16#789C;
   // UNICODE_TO_GBK[23251] := 16#EDD7;
   // UNICODE_TO_GBK[23252] := 16#789D;
   // UNICODE_TO_GBK[23253] := 16#B44D;
   // UNICODE_TO_GBK[23254] := 16#789E;
   // UNICODE_TO_GBK[23255] := 16#B44E;
   // UNICODE_TO_GBK[23256] := 16#789F;
   // UNICODE_TO_GBK[23257] := 16#B5FA;
   // UNICODE_TO_GBK[23258] := 16#78A0;
   // UNICODE_TO_GBK[23259] := 16#B44F;
   // UNICODE_TO_GBK[23260] := 16#78A1;
   // UNICODE_TO_GBK[23261] := 16#EDD8;
   // UNICODE_TO_GBK[23262] := 16#78A2;
   // UNICODE_TO_GBK[23263] := 16#B450;
   // UNICODE_TO_GBK[23264] := 16#78A3;
   // UNICODE_TO_GBK[23265] := 16#EDD9;
   // UNICODE_TO_GBK[23266] := 16#78A4;
   // UNICODE_TO_GBK[23267] := 16#B451;
   // UNICODE_TO_GBK[23268] := 16#78A5;
   // UNICODE_TO_GBK[23269] := 16#EDDC;
   // UNICODE_TO_GBK[23270] := 16#78A6;
   // UNICODE_TO_GBK[23271] := 16#B452;
   // UNICODE_TO_GBK[23272] := 16#78A7;
   // UNICODE_TO_GBK[23273] := 16#B1CC;
   // UNICODE_TO_GBK[23274] := 16#78A8;
   // UNICODE_TO_GBK[23275] := 16#B453;
   // UNICODE_TO_GBK[23276] := 16#78A9;
   // UNICODE_TO_GBK[23277] := 16#B454;
   // UNICODE_TO_GBK[23278] := 16#78AA;
   // UNICODE_TO_GBK[23279] := 16#B455;
   // UNICODE_TO_GBK[23280] := 16#78AB;
   // UNICODE_TO_GBK[23281] := 16#B456;
   // UNICODE_TO_GBK[23282] := 16#78AC;
   // UNICODE_TO_GBK[23283] := 16#B457;
   // UNICODE_TO_GBK[23284] := 16#78AD;
   // UNICODE_TO_GBK[23285] := 16#B458;
   // UNICODE_TO_GBK[23286] := 16#78AE;
   // UNICODE_TO_GBK[23287] := 16#B459;
   // UNICODE_TO_GBK[23288] := 16#78AF;
   // UNICODE_TO_GBK[23289] := 16#B45A;
   // UNICODE_TO_GBK[23290] := 16#78B0;
   // UNICODE_TO_GBK[23291] := 16#C5F6;
   // UNICODE_TO_GBK[23292] := 16#78B1;
   // UNICODE_TO_GBK[23293] := 16#BCEE;
   // UNICODE_TO_GBK[23294] := 16#78B2;
   // UNICODE_TO_GBK[23295] := 16#EDDA;
   // UNICODE_TO_GBK[23296] := 16#78B3;
   // UNICODE_TO_GBK[23297] := 16#CCBC;
   // UNICODE_TO_GBK[23298] := 16#78B4;
   // UNICODE_TO_GBK[23299] := 16#B2EA;
   // UNICODE_TO_GBK[23300] := 16#78B5;
   // UNICODE_TO_GBK[23301] := 16#B45B;
   // UNICODE_TO_GBK[23302] := 16#78B6;
   // UNICODE_TO_GBK[23303] := 16#B45C;
   // UNICODE_TO_GBK[23304] := 16#78B7;
   // UNICODE_TO_GBK[23305] := 16#B45D;
   // UNICODE_TO_GBK[23306] := 16#78B8;
   // UNICODE_TO_GBK[23307] := 16#B45E;
   // UNICODE_TO_GBK[23308] := 16#78B9;
   // UNICODE_TO_GBK[23309] := 16#EDDB;
   // UNICODE_TO_GBK[23310] := 16#78BA;
   // UNICODE_TO_GBK[23311] := 16#B45F;
   // UNICODE_TO_GBK[23312] := 16#78BB;
   // UNICODE_TO_GBK[23313] := 16#B460;
   // UNICODE_TO_GBK[23314] := 16#78BC;
   // UNICODE_TO_GBK[23315] := 16#B461;
   // UNICODE_TO_GBK[23316] := 16#78BD;
   // UNICODE_TO_GBK[23317] := 16#B462;
   // UNICODE_TO_GBK[23318] := 16#78BE;
   // UNICODE_TO_GBK[23319] := 16#C4EB;
   // UNICODE_TO_GBK[23320] := 16#78BF;
   // UNICODE_TO_GBK[23321] := 16#B463;
   // UNICODE_TO_GBK[23322] := 16#78C0;
   // UNICODE_TO_GBK[23323] := 16#B464;
   // UNICODE_TO_GBK[23324] := 16#78C1;
   // UNICODE_TO_GBK[23325] := 16#B4C5;
   // UNICODE_TO_GBK[23326] := 16#78C2;
   // UNICODE_TO_GBK[23327] := 16#B465;
   // UNICODE_TO_GBK[23328] := 16#78C3;
   // UNICODE_TO_GBK[23329] := 16#B466;
   // UNICODE_TO_GBK[23330] := 16#78C4;
   // UNICODE_TO_GBK[23331] := 16#B467;
   // UNICODE_TO_GBK[23332] := 16#78C5;
   // UNICODE_TO_GBK[23333] := 16#B0F5;
   // UNICODE_TO_GBK[23334] := 16#78C6;
   // UNICODE_TO_GBK[23335] := 16#B468;
   // UNICODE_TO_GBK[23336] := 16#78C7;
   // UNICODE_TO_GBK[23337] := 16#B469;
   // UNICODE_TO_GBK[23338] := 16#78C8;
   // UNICODE_TO_GBK[23339] := 16#B46A;
   // UNICODE_TO_GBK[23340] := 16#78C9;
   // UNICODE_TO_GBK[23341] := 16#EDDF;
   // UNICODE_TO_GBK[23342] := 16#78CA;
   // UNICODE_TO_GBK[23343] := 16#C0DA;
   // UNICODE_TO_GBK[23344] := 16#78CB;
   // UNICODE_TO_GBK[23345] := 16#B4E8;
   // UNICODE_TO_GBK[23346] := 16#78CC;
   // UNICODE_TO_GBK[23347] := 16#B46B;
   // UNICODE_TO_GBK[23348] := 16#78CD;
   // UNICODE_TO_GBK[23349] := 16#B46C;
   // UNICODE_TO_GBK[23350] := 16#78CE;
   // UNICODE_TO_GBK[23351] := 16#B46D;
   // UNICODE_TO_GBK[23352] := 16#78CF;
   // UNICODE_TO_GBK[23353] := 16#B46E;
   // UNICODE_TO_GBK[23354] := 16#78D0;
   // UNICODE_TO_GBK[23355] := 16#C5CD;
   // UNICODE_TO_GBK[23356] := 16#78D1;
   // UNICODE_TO_GBK[23357] := 16#B46F;
   // UNICODE_TO_GBK[23358] := 16#78D2;
   // UNICODE_TO_GBK[23359] := 16#B470;
   // UNICODE_TO_GBK[23360] := 16#78D3;
   // UNICODE_TO_GBK[23361] := 16#B471;
   // UNICODE_TO_GBK[23362] := 16#78D4;
   // UNICODE_TO_GBK[23363] := 16#EDDD;
   // UNICODE_TO_GBK[23364] := 16#78D5;
   // UNICODE_TO_GBK[23365] := 16#BFC4;
   // UNICODE_TO_GBK[23366] := 16#78D6;
   // UNICODE_TO_GBK[23367] := 16#B472;
   // UNICODE_TO_GBK[23368] := 16#78D7;
   // UNICODE_TO_GBK[23369] := 16#B473;
   // UNICODE_TO_GBK[23370] := 16#78D8;
   // UNICODE_TO_GBK[23371] := 16#B474;
   // UNICODE_TO_GBK[23372] := 16#78D9;
   // UNICODE_TO_GBK[23373] := 16#EDDE;
   // UNICODE_TO_GBK[23374] := 16#78DA;
   // UNICODE_TO_GBK[23375] := 16#B475;
   // UNICODE_TO_GBK[23376] := 16#78DB;
   // UNICODE_TO_GBK[23377] := 16#B476;
   // UNICODE_TO_GBK[23378] := 16#78DC;
   // UNICODE_TO_GBK[23379] := 16#B477;
   // UNICODE_TO_GBK[23380] := 16#78DD;
   // UNICODE_TO_GBK[23381] := 16#B478;
   // UNICODE_TO_GBK[23382] := 16#78DE;
   // UNICODE_TO_GBK[23383] := 16#B479;
   // UNICODE_TO_GBK[23384] := 16#78DF;
   // UNICODE_TO_GBK[23385] := 16#B47A;
   // UNICODE_TO_GBK[23386] := 16#78E0;
   // UNICODE_TO_GBK[23387] := 16#B47B;
   // UNICODE_TO_GBK[23388] := 16#78E1;
   // UNICODE_TO_GBK[23389] := 16#B47C;
   // UNICODE_TO_GBK[23390] := 16#78E2;
   // UNICODE_TO_GBK[23391] := 16#B47D;
   // UNICODE_TO_GBK[23392] := 16#78E3;
   // UNICODE_TO_GBK[23393] := 16#B47E;
   // UNICODE_TO_GBK[23394] := 16#78E4;
   // UNICODE_TO_GBK[23395] := 16#B480;
   // UNICODE_TO_GBK[23396] := 16#78E5;
   // UNICODE_TO_GBK[23397] := 16#B481;
   // UNICODE_TO_GBK[23398] := 16#78E6;
   // UNICODE_TO_GBK[23399] := 16#B482;
   // UNICODE_TO_GBK[23400] := 16#78E7;
   // UNICODE_TO_GBK[23401] := 16#B483;
   // UNICODE_TO_GBK[23402] := 16#78E8;
   // UNICODE_TO_GBK[23403] := 16#C4A5;
   // UNICODE_TO_GBK[23404] := 16#78E9;
   // UNICODE_TO_GBK[23405] := 16#B484;
   // UNICODE_TO_GBK[23406] := 16#78EA;
   // UNICODE_TO_GBK[23407] := 16#B485;
   // UNICODE_TO_GBK[23408] := 16#78EB;
   // UNICODE_TO_GBK[23409] := 16#B486;
   // UNICODE_TO_GBK[23410] := 16#78EC;
   // UNICODE_TO_GBK[23411] := 16#EDE0;
   // UNICODE_TO_GBK[23412] := 16#78ED;
   // UNICODE_TO_GBK[23413] := 16#B487;
   // UNICODE_TO_GBK[23414] := 16#78EE;
   // UNICODE_TO_GBK[23415] := 16#B488;
   // UNICODE_TO_GBK[23416] := 16#78EF;
   // UNICODE_TO_GBK[23417] := 16#B489;
   // UNICODE_TO_GBK[23418] := 16#78F0;
   // UNICODE_TO_GBK[23419] := 16#B48A;
   // UNICODE_TO_GBK[23420] := 16#78F1;
   // UNICODE_TO_GBK[23421] := 16#B48B;
   // UNICODE_TO_GBK[23422] := 16#78F2;
   // UNICODE_TO_GBK[23423] := 16#EDE1;
   // UNICODE_TO_GBK[23424] := 16#78F3;
   // UNICODE_TO_GBK[23425] := 16#B48C;
   // UNICODE_TO_GBK[23426] := 16#78F4;
   // UNICODE_TO_GBK[23427] := 16#EDE3;
   // UNICODE_TO_GBK[23428] := 16#78F5;
   // UNICODE_TO_GBK[23429] := 16#B48D;
   // UNICODE_TO_GBK[23430] := 16#78F6;
   // UNICODE_TO_GBK[23431] := 16#B48E;
   // UNICODE_TO_GBK[23432] := 16#78F7;
   // UNICODE_TO_GBK[23433] := 16#C1D7;
   // UNICODE_TO_GBK[23434] := 16#78F8;
   // UNICODE_TO_GBK[23435] := 16#B48F;
   // UNICODE_TO_GBK[23436] := 16#78F9;
   // UNICODE_TO_GBK[23437] := 16#B490;
   // UNICODE_TO_GBK[23438] := 16#78FA;
   // UNICODE_TO_GBK[23439] := 16#BBC7;
   // UNICODE_TO_GBK[23440] := 16#78FB;
   // UNICODE_TO_GBK[23441] := 16#B491;
   // UNICODE_TO_GBK[23442] := 16#78FC;
   // UNICODE_TO_GBK[23443] := 16#B492;
   // UNICODE_TO_GBK[23444] := 16#78FD;
   // UNICODE_TO_GBK[23445] := 16#B493;
   // UNICODE_TO_GBK[23446] := 16#78FE;
   // UNICODE_TO_GBK[23447] := 16#B494;
   // UNICODE_TO_GBK[23448] := 16#78FF;
   // UNICODE_TO_GBK[23449] := 16#B495;
   // UNICODE_TO_GBK[23450] := 16#7900;
   // UNICODE_TO_GBK[23451] := 16#B496;
   // UNICODE_TO_GBK[23452] := 16#7901;
   // UNICODE_TO_GBK[23453] := 16#BDB8;
   // UNICODE_TO_GBK[23454] := 16#7902;
   // UNICODE_TO_GBK[23455] := 16#B497;
   // UNICODE_TO_GBK[23456] := 16#7903;
   // UNICODE_TO_GBK[23457] := 16#B498;
   // UNICODE_TO_GBK[23458] := 16#7904;
   // UNICODE_TO_GBK[23459] := 16#B499;
   // UNICODE_TO_GBK[23460] := 16#7905;
   // UNICODE_TO_GBK[23461] := 16#EDE2;
   // UNICODE_TO_GBK[23462] := 16#7906;
   // UNICODE_TO_GBK[23463] := 16#B49A;
   // UNICODE_TO_GBK[23464] := 16#7907;
   // UNICODE_TO_GBK[23465] := 16#B49B;
   // UNICODE_TO_GBK[23466] := 16#7908;
   // UNICODE_TO_GBK[23467] := 16#B49C;
   // UNICODE_TO_GBK[23468] := 16#7909;
   // UNICODE_TO_GBK[23469] := 16#B49D;
   // UNICODE_TO_GBK[23470] := 16#790A;
   // UNICODE_TO_GBK[23471] := 16#B49E;
   // UNICODE_TO_GBK[23472] := 16#790B;
   // UNICODE_TO_GBK[23473] := 16#B49F;
   // UNICODE_TO_GBK[23474] := 16#790C;
   // UNICODE_TO_GBK[23475] := 16#B4A0;
   // UNICODE_TO_GBK[23476] := 16#790D;
   // UNICODE_TO_GBK[23477] := 16#B540;
   // UNICODE_TO_GBK[23478] := 16#790E;
   // UNICODE_TO_GBK[23479] := 16#B541;
   // UNICODE_TO_GBK[23480] := 16#790F;
   // UNICODE_TO_GBK[23481] := 16#B542;
   // UNICODE_TO_GBK[23482] := 16#7910;
   // UNICODE_TO_GBK[23483] := 16#B543;
   // UNICODE_TO_GBK[23484] := 16#7911;
   // UNICODE_TO_GBK[23485] := 16#B544;
   // UNICODE_TO_GBK[23486] := 16#7912;
   // UNICODE_TO_GBK[23487] := 16#B545;
   // UNICODE_TO_GBK[23488] := 16#7913;
   // UNICODE_TO_GBK[23489] := 16#EDE4;
   // UNICODE_TO_GBK[23490] := 16#7914;
   // UNICODE_TO_GBK[23491] := 16#B546;
   // UNICODE_TO_GBK[23492] := 16#7915;
   // UNICODE_TO_GBK[23493] := 16#B547;
   // UNICODE_TO_GBK[23494] := 16#7916;
   // UNICODE_TO_GBK[23495] := 16#B548;
   // UNICODE_TO_GBK[23496] := 16#7917;
   // UNICODE_TO_GBK[23497] := 16#B549;
   // UNICODE_TO_GBK[23498] := 16#7918;
   // UNICODE_TO_GBK[23499] := 16#B54A;
   // UNICODE_TO_GBK[23500] := 16#7919;
   // UNICODE_TO_GBK[23501] := 16#B54B;
   // UNICODE_TO_GBK[23502] := 16#791A;
   // UNICODE_TO_GBK[23503] := 16#B54C;
   // UNICODE_TO_GBK[23504] := 16#791B;
   // UNICODE_TO_GBK[23505] := 16#B54D;
   // UNICODE_TO_GBK[23506] := 16#791C;
   // UNICODE_TO_GBK[23507] := 16#B54E;
   // UNICODE_TO_GBK[23508] := 16#791D;
   // UNICODE_TO_GBK[23509] := 16#B54F;
   // UNICODE_TO_GBK[23510] := 16#791E;
   // UNICODE_TO_GBK[23511] := 16#EDE6;
   // UNICODE_TO_GBK[23512] := 16#791F;
   // UNICODE_TO_GBK[23513] := 16#B550;
   // UNICODE_TO_GBK[23514] := 16#7920;
   // UNICODE_TO_GBK[23515] := 16#B551;
   // UNICODE_TO_GBK[23516] := 16#7921;
   // UNICODE_TO_GBK[23517] := 16#B552;
   // UNICODE_TO_GBK[23518] := 16#7922;
   // UNICODE_TO_GBK[23519] := 16#B553;
   // UNICODE_TO_GBK[23520] := 16#7923;
   // UNICODE_TO_GBK[23521] := 16#B554;
   // UNICODE_TO_GBK[23522] := 16#7924;
   // UNICODE_TO_GBK[23523] := 16#EDE5;
   // UNICODE_TO_GBK[23524] := 16#7925;
   // UNICODE_TO_GBK[23525] := 16#B555;
   // UNICODE_TO_GBK[23526] := 16#7926;
   // UNICODE_TO_GBK[23527] := 16#B556;
   // UNICODE_TO_GBK[23528] := 16#7927;
   // UNICODE_TO_GBK[23529] := 16#B557;
   // UNICODE_TO_GBK[23530] := 16#7928;
   // UNICODE_TO_GBK[23531] := 16#B558;
   // UNICODE_TO_GBK[23532] := 16#7929;
   // UNICODE_TO_GBK[23533] := 16#B559;
   // UNICODE_TO_GBK[23534] := 16#792A;
   // UNICODE_TO_GBK[23535] := 16#B55A;
   // UNICODE_TO_GBK[23536] := 16#792B;
   // UNICODE_TO_GBK[23537] := 16#B55B;
   // UNICODE_TO_GBK[23538] := 16#792C;
   // UNICODE_TO_GBK[23539] := 16#B55C;
   // UNICODE_TO_GBK[23540] := 16#792D;
   // UNICODE_TO_GBK[23541] := 16#B55D;
   // UNICODE_TO_GBK[23542] := 16#792E;
   // UNICODE_TO_GBK[23543] := 16#B55E;
   // UNICODE_TO_GBK[23544] := 16#792F;
   // UNICODE_TO_GBK[23545] := 16#B55F;
   // UNICODE_TO_GBK[23546] := 16#7930;
   // UNICODE_TO_GBK[23547] := 16#B560;
   // UNICODE_TO_GBK[23548] := 16#7931;
   // UNICODE_TO_GBK[23549] := 16#B561;
   // UNICODE_TO_GBK[23550] := 16#7932;
   // UNICODE_TO_GBK[23551] := 16#B562;
   // UNICODE_TO_GBK[23552] := 16#7933;
   // UNICODE_TO_GBK[23553] := 16#B563;
   // UNICODE_TO_GBK[23554] := 16#7934;
   // UNICODE_TO_GBK[23555] := 16#EDE7;
   // UNICODE_TO_GBK[23556] := 16#7935;
   // UNICODE_TO_GBK[23557] := 16#B564;
   // UNICODE_TO_GBK[23558] := 16#7936;
   // UNICODE_TO_GBK[23559] := 16#B565;
   // UNICODE_TO_GBK[23560] := 16#7937;
   // UNICODE_TO_GBK[23561] := 16#B566;
   // UNICODE_TO_GBK[23562] := 16#7938;
   // UNICODE_TO_GBK[23563] := 16#B567;
   // UNICODE_TO_GBK[23564] := 16#7939;
   // UNICODE_TO_GBK[23565] := 16#B568;
   // UNICODE_TO_GBK[23566] := 16#793A;
   // UNICODE_TO_GBK[23567] := 16#CABE;
   // UNICODE_TO_GBK[23568] := 16#793B;
   // UNICODE_TO_GBK[23569] := 16#ECEA;
   // UNICODE_TO_GBK[23570] := 16#793C;
   // UNICODE_TO_GBK[23571] := 16#C0F1;
   // UNICODE_TO_GBK[23572] := 16#793D;
   // UNICODE_TO_GBK[23573] := 16#B569;
   // UNICODE_TO_GBK[23574] := 16#793E;
   // UNICODE_TO_GBK[23575] := 16#C9E7;
   // UNICODE_TO_GBK[23576] := 16#793F;
   // UNICODE_TO_GBK[23577] := 16#B56A;
   // UNICODE_TO_GBK[23578] := 16#7940;
   // UNICODE_TO_GBK[23579] := 16#ECEB;
   // UNICODE_TO_GBK[23580] := 16#7941;
   // UNICODE_TO_GBK[23581] := 16#C6EE;
   // UNICODE_TO_GBK[23582] := 16#7942;
   // UNICODE_TO_GBK[23583] := 16#B56B;
   // UNICODE_TO_GBK[23584] := 16#7943;
   // UNICODE_TO_GBK[23585] := 16#B56C;
   // UNICODE_TO_GBK[23586] := 16#7944;
   // UNICODE_TO_GBK[23587] := 16#B56D;
   // UNICODE_TO_GBK[23588] := 16#7945;
   // UNICODE_TO_GBK[23589] := 16#B56E;
   // UNICODE_TO_GBK[23590] := 16#7946;
   // UNICODE_TO_GBK[23591] := 16#ECEC;
   // UNICODE_TO_GBK[23592] := 16#7947;
   // UNICODE_TO_GBK[23593] := 16#B56F;
   // UNICODE_TO_GBK[23594] := 16#7948;
   // UNICODE_TO_GBK[23595] := 16#C6ED;
   // UNICODE_TO_GBK[23596] := 16#7949;
   // UNICODE_TO_GBK[23597] := 16#ECED;
   // UNICODE_TO_GBK[23598] := 16#794A;
   // UNICODE_TO_GBK[23599] := 16#B570;
   // UNICODE_TO_GBK[23600] := 16#794B;
   // UNICODE_TO_GBK[23601] := 16#B571;
   // UNICODE_TO_GBK[23602] := 16#794C;
   // UNICODE_TO_GBK[23603] := 16#B572;
   // UNICODE_TO_GBK[23604] := 16#794D;
   // UNICODE_TO_GBK[23605] := 16#B573;
   // UNICODE_TO_GBK[23606] := 16#794E;
   // UNICODE_TO_GBK[23607] := 16#B574;
   // UNICODE_TO_GBK[23608] := 16#794F;
   // UNICODE_TO_GBK[23609] := 16#B575;
   // UNICODE_TO_GBK[23610] := 16#7950;
   // UNICODE_TO_GBK[23611] := 16#B576;
   // UNICODE_TO_GBK[23612] := 16#7951;
   // UNICODE_TO_GBK[23613] := 16#B577;
   // UNICODE_TO_GBK[23614] := 16#7952;
   // UNICODE_TO_GBK[23615] := 16#B578;
   // UNICODE_TO_GBK[23616] := 16#7953;
   // UNICODE_TO_GBK[23617] := 16#ECF0;
   // UNICODE_TO_GBK[23618] := 16#7954;
   // UNICODE_TO_GBK[23619] := 16#B579;
   // UNICODE_TO_GBK[23620] := 16#7955;
   // UNICODE_TO_GBK[23621] := 16#B57A;
   // UNICODE_TO_GBK[23622] := 16#7956;
   // UNICODE_TO_GBK[23623] := 16#D7E6;
   // UNICODE_TO_GBK[23624] := 16#7957;
   // UNICODE_TO_GBK[23625] := 16#ECF3;
   // UNICODE_TO_GBK[23626] := 16#7958;
   // UNICODE_TO_GBK[23627] := 16#B57B;
   // UNICODE_TO_GBK[23628] := 16#7959;
   // UNICODE_TO_GBK[23629] := 16#B57C;
   // UNICODE_TO_GBK[23630] := 16#795A;
   // UNICODE_TO_GBK[23631] := 16#ECF1;
   // UNICODE_TO_GBK[23632] := 16#795B;
   // UNICODE_TO_GBK[23633] := 16#ECEE;
   // UNICODE_TO_GBK[23634] := 16#795C;
   // UNICODE_TO_GBK[23635] := 16#ECEF;
   // UNICODE_TO_GBK[23636] := 16#795D;
   // UNICODE_TO_GBK[23637] := 16#D7A3;
   // UNICODE_TO_GBK[23638] := 16#795E;
   // UNICODE_TO_GBK[23639] := 16#C9F1;
   // UNICODE_TO_GBK[23640] := 16#795F;
   // UNICODE_TO_GBK[23641] := 16#CBEE;
   // UNICODE_TO_GBK[23642] := 16#7960;
   // UNICODE_TO_GBK[23643] := 16#ECF4;
   // UNICODE_TO_GBK[23644] := 16#7961;
   // UNICODE_TO_GBK[23645] := 16#B57D;
   // UNICODE_TO_GBK[23646] := 16#7962;
   // UNICODE_TO_GBK[23647] := 16#ECF2;
   // UNICODE_TO_GBK[23648] := 16#7963;
   // UNICODE_TO_GBK[23649] := 16#B57E;
   // UNICODE_TO_GBK[23650] := 16#7964;
   // UNICODE_TO_GBK[23651] := 16#B580;
   // UNICODE_TO_GBK[23652] := 16#7965;
   // UNICODE_TO_GBK[23653] := 16#CFE9;
   // UNICODE_TO_GBK[23654] := 16#7966;
   // UNICODE_TO_GBK[23655] := 16#B581;
   // UNICODE_TO_GBK[23656] := 16#7967;
   // UNICODE_TO_GBK[23657] := 16#ECF6;
   // UNICODE_TO_GBK[23658] := 16#7968;
   // UNICODE_TO_GBK[23659] := 16#C6B1;
   // UNICODE_TO_GBK[23660] := 16#7969;
   // UNICODE_TO_GBK[23661] := 16#B582;
   // UNICODE_TO_GBK[23662] := 16#796A;
   // UNICODE_TO_GBK[23663] := 16#B583;
   // UNICODE_TO_GBK[23664] := 16#796B;
   // UNICODE_TO_GBK[23665] := 16#B584;
   // UNICODE_TO_GBK[23666] := 16#796C;
   // UNICODE_TO_GBK[23667] := 16#B585;
   // UNICODE_TO_GBK[23668] := 16#796D;
   // UNICODE_TO_GBK[23669] := 16#BCC0;
   // UNICODE_TO_GBK[23670] := 16#796E;
   // UNICODE_TO_GBK[23671] := 16#B586;
   // UNICODE_TO_GBK[23672] := 16#796F;
   // UNICODE_TO_GBK[23673] := 16#ECF5;
   // UNICODE_TO_GBK[23674] := 16#7970;
   // UNICODE_TO_GBK[23675] := 16#B587;
   // UNICODE_TO_GBK[23676] := 16#7971;
   // UNICODE_TO_GBK[23677] := 16#B588;
   // UNICODE_TO_GBK[23678] := 16#7972;
   // UNICODE_TO_GBK[23679] := 16#B589;
   // UNICODE_TO_GBK[23680] := 16#7973;
   // UNICODE_TO_GBK[23681] := 16#B58A;
   // UNICODE_TO_GBK[23682] := 16#7974;
   // UNICODE_TO_GBK[23683] := 16#B58B;
   // UNICODE_TO_GBK[23684] := 16#7975;
   // UNICODE_TO_GBK[23685] := 16#B58C;
   // UNICODE_TO_GBK[23686] := 16#7976;
   // UNICODE_TO_GBK[23687] := 16#B58D;
   // UNICODE_TO_GBK[23688] := 16#7977;
   // UNICODE_TO_GBK[23689] := 16#B5BB;
   // UNICODE_TO_GBK[23690] := 16#7978;
   // UNICODE_TO_GBK[23691] := 16#BBF6;
   // UNICODE_TO_GBK[23692] := 16#7979;
   // UNICODE_TO_GBK[23693] := 16#B58E;
   // UNICODE_TO_GBK[23694] := 16#797A;
   // UNICODE_TO_GBK[23695] := 16#ECF7;
   // UNICODE_TO_GBK[23696] := 16#797B;
   // UNICODE_TO_GBK[23697] := 16#B58F;
   // UNICODE_TO_GBK[23698] := 16#797C;
   // UNICODE_TO_GBK[23699] := 16#B590;
   // UNICODE_TO_GBK[23700] := 16#797D;
   // UNICODE_TO_GBK[23701] := 16#B591;
   // UNICODE_TO_GBK[23702] := 16#797E;
   // UNICODE_TO_GBK[23703] := 16#B592;
   // UNICODE_TO_GBK[23704] := 16#797F;
   // UNICODE_TO_GBK[23705] := 16#B593;
   // UNICODE_TO_GBK[23706] := 16#7980;
   // UNICODE_TO_GBK[23707] := 16#D9F7;
   // UNICODE_TO_GBK[23708] := 16#7981;
   // UNICODE_TO_GBK[23709] := 16#BDFB;
   // UNICODE_TO_GBK[23710] := 16#7982;
   // UNICODE_TO_GBK[23711] := 16#B594;
   // UNICODE_TO_GBK[23712] := 16#7983;
   // UNICODE_TO_GBK[23713] := 16#B595;
   // UNICODE_TO_GBK[23714] := 16#7984;
   // UNICODE_TO_GBK[23715] := 16#C2BB;
   // UNICODE_TO_GBK[23716] := 16#7985;
   // UNICODE_TO_GBK[23717] := 16#ECF8;
   // UNICODE_TO_GBK[23718] := 16#7986;
   // UNICODE_TO_GBK[23719] := 16#B596;
   // UNICODE_TO_GBK[23720] := 16#7987;
   // UNICODE_TO_GBK[23721] := 16#B597;
   // UNICODE_TO_GBK[23722] := 16#7988;
   // UNICODE_TO_GBK[23723] := 16#B598;
   // UNICODE_TO_GBK[23724] := 16#7989;
   // UNICODE_TO_GBK[23725] := 16#B599;
   // UNICODE_TO_GBK[23726] := 16#798A;
   // UNICODE_TO_GBK[23727] := 16#ECF9;
   // UNICODE_TO_GBK[23728] := 16#798B;
   // UNICODE_TO_GBK[23729] := 16#B59A;
   // UNICODE_TO_GBK[23730] := 16#798C;
   // UNICODE_TO_GBK[23731] := 16#B59B;
   // UNICODE_TO_GBK[23732] := 16#798D;
   // UNICODE_TO_GBK[23733] := 16#B59C;
   // UNICODE_TO_GBK[23734] := 16#798E;
   // UNICODE_TO_GBK[23735] := 16#B59D;
   // UNICODE_TO_GBK[23736] := 16#798F;
   // UNICODE_TO_GBK[23737] := 16#B8A3;
   // UNICODE_TO_GBK[23738] := 16#7990;
   // UNICODE_TO_GBK[23739] := 16#B59E;
   // UNICODE_TO_GBK[23740] := 16#7991;
   // UNICODE_TO_GBK[23741] := 16#B59F;
   // UNICODE_TO_GBK[23742] := 16#7992;
   // UNICODE_TO_GBK[23743] := 16#B5A0;
   // UNICODE_TO_GBK[23744] := 16#7993;
   // UNICODE_TO_GBK[23745] := 16#B640;
   // UNICODE_TO_GBK[23746] := 16#7994;
   // UNICODE_TO_GBK[23747] := 16#B641;
   // UNICODE_TO_GBK[23748] := 16#7995;
   // UNICODE_TO_GBK[23749] := 16#B642;
   // UNICODE_TO_GBK[23750] := 16#7996;
   // UNICODE_TO_GBK[23751] := 16#B643;
   // UNICODE_TO_GBK[23752] := 16#7997;
   // UNICODE_TO_GBK[23753] := 16#B644;
   // UNICODE_TO_GBK[23754] := 16#7998;
   // UNICODE_TO_GBK[23755] := 16#B645;
   // UNICODE_TO_GBK[23756] := 16#7999;
   // UNICODE_TO_GBK[23757] := 16#B646;
   // UNICODE_TO_GBK[23758] := 16#799A;
   // UNICODE_TO_GBK[23759] := 16#ECFA;
   // UNICODE_TO_GBK[23760] := 16#799B;
   // UNICODE_TO_GBK[23761] := 16#B647;
   // UNICODE_TO_GBK[23762] := 16#799C;
   // UNICODE_TO_GBK[23763] := 16#B648;
   // UNICODE_TO_GBK[23764] := 16#799D;
   // UNICODE_TO_GBK[23765] := 16#B649;
   // UNICODE_TO_GBK[23766] := 16#799E;
   // UNICODE_TO_GBK[23767] := 16#B64A;
   // UNICODE_TO_GBK[23768] := 16#799F;
   // UNICODE_TO_GBK[23769] := 16#B64B;
   // UNICODE_TO_GBK[23770] := 16#79A0;
   // UNICODE_TO_GBK[23771] := 16#B64C;
   // UNICODE_TO_GBK[23772] := 16#79A1;
   // UNICODE_TO_GBK[23773] := 16#B64D;
   // UNICODE_TO_GBK[23774] := 16#79A2;
   // UNICODE_TO_GBK[23775] := 16#B64E;
   // UNICODE_TO_GBK[23776] := 16#79A3;
   // UNICODE_TO_GBK[23777] := 16#B64F;
   // UNICODE_TO_GBK[23778] := 16#79A4;
   // UNICODE_TO_GBK[23779] := 16#B650;
   // UNICODE_TO_GBK[23780] := 16#79A5;
   // UNICODE_TO_GBK[23781] := 16#B651;
   // UNICODE_TO_GBK[23782] := 16#79A6;
   // UNICODE_TO_GBK[23783] := 16#B652;
   // UNICODE_TO_GBK[23784] := 16#79A7;
   // UNICODE_TO_GBK[23785] := 16#ECFB;
   // UNICODE_TO_GBK[23786] := 16#79A8;
   // UNICODE_TO_GBK[23787] := 16#B653;
   // UNICODE_TO_GBK[23788] := 16#79A9;
   // UNICODE_TO_GBK[23789] := 16#B654;
   // UNICODE_TO_GBK[23790] := 16#79AA;
   // UNICODE_TO_GBK[23791] := 16#B655;
   // UNICODE_TO_GBK[23792] := 16#79AB;
   // UNICODE_TO_GBK[23793] := 16#B656;
   // UNICODE_TO_GBK[23794] := 16#79AC;
   // UNICODE_TO_GBK[23795] := 16#B657;
   // UNICODE_TO_GBK[23796] := 16#79AD;
   // UNICODE_TO_GBK[23797] := 16#B658;
   // UNICODE_TO_GBK[23798] := 16#79AE;
   // UNICODE_TO_GBK[23799] := 16#B659;
   // UNICODE_TO_GBK[23800] := 16#79AF;
   // UNICODE_TO_GBK[23801] := 16#B65A;
   // UNICODE_TO_GBK[23802] := 16#79B0;
   // UNICODE_TO_GBK[23803] := 16#B65B;
   // UNICODE_TO_GBK[23804] := 16#79B1;
   // UNICODE_TO_GBK[23805] := 16#B65C;
   // UNICODE_TO_GBK[23806] := 16#79B2;
   // UNICODE_TO_GBK[23807] := 16#B65D;
   // UNICODE_TO_GBK[23808] := 16#79B3;
   // UNICODE_TO_GBK[23809] := 16#ECFC;
   // UNICODE_TO_GBK[23810] := 16#79B4;
   // UNICODE_TO_GBK[23811] := 16#B65E;
   // UNICODE_TO_GBK[23812] := 16#79B5;
   // UNICODE_TO_GBK[23813] := 16#B65F;
   // UNICODE_TO_GBK[23814] := 16#79B6;
   // UNICODE_TO_GBK[23815] := 16#B660;
   // UNICODE_TO_GBK[23816] := 16#79B7;
   // UNICODE_TO_GBK[23817] := 16#B661;
   // UNICODE_TO_GBK[23818] := 16#79B8;
   // UNICODE_TO_GBK[23819] := 16#B662;
   // UNICODE_TO_GBK[23820] := 16#79B9;
   // UNICODE_TO_GBK[23821] := 16#D3ED;
   // UNICODE_TO_GBK[23822] := 16#79BA;
   // UNICODE_TO_GBK[23823] := 16#D8AE;
   // UNICODE_TO_GBK[23824] := 16#79BB;
   // UNICODE_TO_GBK[23825] := 16#C0EB;
   // UNICODE_TO_GBK[23826] := 16#79BC;
   // UNICODE_TO_GBK[23827] := 16#B663;
   // UNICODE_TO_GBK[23828] := 16#79BD;
   // UNICODE_TO_GBK[23829] := 16#C7DD;
   // UNICODE_TO_GBK[23830] := 16#79BE;
   // UNICODE_TO_GBK[23831] := 16#BACC;
   // UNICODE_TO_GBK[23832] := 16#79BF;
   // UNICODE_TO_GBK[23833] := 16#B664;
   // UNICODE_TO_GBK[23834] := 16#79C0;
   // UNICODE_TO_GBK[23835] := 16#D0E3;
   // UNICODE_TO_GBK[23836] := 16#79C1;
   // UNICODE_TO_GBK[23837] := 16#CBBD;
   // UNICODE_TO_GBK[23838] := 16#79C2;
   // UNICODE_TO_GBK[23839] := 16#B665;
   // UNICODE_TO_GBK[23840] := 16#79C3;
   // UNICODE_TO_GBK[23841] := 16#CDBA;
   // UNICODE_TO_GBK[23842] := 16#79C4;
   // UNICODE_TO_GBK[23843] := 16#B666;
   // UNICODE_TO_GBK[23844] := 16#79C5;
   // UNICODE_TO_GBK[23845] := 16#B667;
   // UNICODE_TO_GBK[23846] := 16#79C6;
   // UNICODE_TO_GBK[23847] := 16#B8D1;
   // UNICODE_TO_GBK[23848] := 16#79C7;
   // UNICODE_TO_GBK[23849] := 16#B668;
   // UNICODE_TO_GBK[23850] := 16#79C8;
   // UNICODE_TO_GBK[23851] := 16#B669;
   // UNICODE_TO_GBK[23852] := 16#79C9;
   // UNICODE_TO_GBK[23853] := 16#B1FC;
   // UNICODE_TO_GBK[23854] := 16#79CA;
   // UNICODE_TO_GBK[23855] := 16#B66A;
   // UNICODE_TO_GBK[23856] := 16#79CB;
   // UNICODE_TO_GBK[23857] := 16#C7EF;
   // UNICODE_TO_GBK[23858] := 16#79CC;
   // UNICODE_TO_GBK[23859] := 16#B66B;
   // UNICODE_TO_GBK[23860] := 16#79CD;
   // UNICODE_TO_GBK[23861] := 16#D6D6;
   // UNICODE_TO_GBK[23862] := 16#79CE;
   // UNICODE_TO_GBK[23863] := 16#B66C;
   // UNICODE_TO_GBK[23864] := 16#79CF;
   // UNICODE_TO_GBK[23865] := 16#B66D;
   // UNICODE_TO_GBK[23866] := 16#79D0;
   // UNICODE_TO_GBK[23867] := 16#B66E;
   // UNICODE_TO_GBK[23868] := 16#79D1;
   // UNICODE_TO_GBK[23869] := 16#BFC6;
   // UNICODE_TO_GBK[23870] := 16#79D2;
   // UNICODE_TO_GBK[23871] := 16#C3EB;
   // UNICODE_TO_GBK[23872] := 16#79D3;
   // UNICODE_TO_GBK[23873] := 16#B66F;
   // UNICODE_TO_GBK[23874] := 16#79D4;
   // UNICODE_TO_GBK[23875] := 16#B670;
   // UNICODE_TO_GBK[23876] := 16#79D5;
   // UNICODE_TO_GBK[23877] := 16#EFF5;
   // UNICODE_TO_GBK[23878] := 16#79D6;
   // UNICODE_TO_GBK[23879] := 16#B671;
   // UNICODE_TO_GBK[23880] := 16#79D7;
   // UNICODE_TO_GBK[23881] := 16#B672;
   // UNICODE_TO_GBK[23882] := 16#79D8;
   // UNICODE_TO_GBK[23883] := 16#C3D8;
   // UNICODE_TO_GBK[23884] := 16#79D9;
   // UNICODE_TO_GBK[23885] := 16#B673;
   // UNICODE_TO_GBK[23886] := 16#79DA;
   // UNICODE_TO_GBK[23887] := 16#B674;
   // UNICODE_TO_GBK[23888] := 16#79DB;
   // UNICODE_TO_GBK[23889] := 16#B675;
   // UNICODE_TO_GBK[23890] := 16#79DC;
   // UNICODE_TO_GBK[23891] := 16#B676;
   // UNICODE_TO_GBK[23892] := 16#79DD;
   // UNICODE_TO_GBK[23893] := 16#B677;
   // UNICODE_TO_GBK[23894] := 16#79DE;
   // UNICODE_TO_GBK[23895] := 16#B678;
   // UNICODE_TO_GBK[23896] := 16#79DF;
   // UNICODE_TO_GBK[23897] := 16#D7E2;
   // UNICODE_TO_GBK[23898] := 16#79E0;
   // UNICODE_TO_GBK[23899] := 16#B679;
   // UNICODE_TO_GBK[23900] := 16#79E1;
   // UNICODE_TO_GBK[23901] := 16#B67A;
   // UNICODE_TO_GBK[23902] := 16#79E2;
   // UNICODE_TO_GBK[23903] := 16#B67B;
   // UNICODE_TO_GBK[23904] := 16#79E3;
   // UNICODE_TO_GBK[23905] := 16#EFF7;
   // UNICODE_TO_GBK[23906] := 16#79E4;
   // UNICODE_TO_GBK[23907] := 16#B3D3;
   // UNICODE_TO_GBK[23908] := 16#79E5;
   // UNICODE_TO_GBK[23909] := 16#B67C;
   // UNICODE_TO_GBK[23910] := 16#79E6;
   // UNICODE_TO_GBK[23911] := 16#C7D8;
   // UNICODE_TO_GBK[23912] := 16#79E7;
   // UNICODE_TO_GBK[23913] := 16#D1ED;
   // UNICODE_TO_GBK[23914] := 16#79E8;
   // UNICODE_TO_GBK[23915] := 16#B67D;
   // UNICODE_TO_GBK[23916] := 16#79E9;
   // UNICODE_TO_GBK[23917] := 16#D6C8;
   // UNICODE_TO_GBK[23918] := 16#79EA;
   // UNICODE_TO_GBK[23919] := 16#B67E;
   // UNICODE_TO_GBK[23920] := 16#79EB;
   // UNICODE_TO_GBK[23921] := 16#EFF8;
   // UNICODE_TO_GBK[23922] := 16#79EC;
   // UNICODE_TO_GBK[23923] := 16#B680;
   // UNICODE_TO_GBK[23924] := 16#79ED;
   // UNICODE_TO_GBK[23925] := 16#EFF6;
   // UNICODE_TO_GBK[23926] := 16#79EE;
   // UNICODE_TO_GBK[23927] := 16#B681;
   // UNICODE_TO_GBK[23928] := 16#79EF;
   // UNICODE_TO_GBK[23929] := 16#BBFD;
   // UNICODE_TO_GBK[23930] := 16#79F0;
   // UNICODE_TO_GBK[23931] := 16#B3C6;
   // UNICODE_TO_GBK[23932] := 16#79F1;
   // UNICODE_TO_GBK[23933] := 16#B682;
   // UNICODE_TO_GBK[23934] := 16#79F2;
   // UNICODE_TO_GBK[23935] := 16#B683;
   // UNICODE_TO_GBK[23936] := 16#79F3;
   // UNICODE_TO_GBK[23937] := 16#B684;
   // UNICODE_TO_GBK[23938] := 16#79F4;
   // UNICODE_TO_GBK[23939] := 16#B685;
   // UNICODE_TO_GBK[23940] := 16#79F5;
   // UNICODE_TO_GBK[23941] := 16#B686;
   // UNICODE_TO_GBK[23942] := 16#79F6;
   // UNICODE_TO_GBK[23943] := 16#B687;
   // UNICODE_TO_GBK[23944] := 16#79F7;
   // UNICODE_TO_GBK[23945] := 16#B688;
   // UNICODE_TO_GBK[23946] := 16#79F8;
   // UNICODE_TO_GBK[23947] := 16#BDD5;
   // UNICODE_TO_GBK[23948] := 16#79F9;
   // UNICODE_TO_GBK[23949] := 16#B689;
   // UNICODE_TO_GBK[23950] := 16#79FA;
   // UNICODE_TO_GBK[23951] := 16#B68A;
   // UNICODE_TO_GBK[23952] := 16#79FB;
   // UNICODE_TO_GBK[23953] := 16#D2C6;
   // UNICODE_TO_GBK[23954] := 16#79FC;
   // UNICODE_TO_GBK[23955] := 16#B68B;
   // UNICODE_TO_GBK[23956] := 16#79FD;
   // UNICODE_TO_GBK[23957] := 16#BBE0;
   // UNICODE_TO_GBK[23958] := 16#79FE;
   // UNICODE_TO_GBK[23959] := 16#B68C;
   // UNICODE_TO_GBK[23960] := 16#79FF;
   // UNICODE_TO_GBK[23961] := 16#B68D;
   // UNICODE_TO_GBK[23962] := 16#7A00;
   // UNICODE_TO_GBK[23963] := 16#CFA1;
   // UNICODE_TO_GBK[23964] := 16#7A01;
   // UNICODE_TO_GBK[23965] := 16#B68E;
   // UNICODE_TO_GBK[23966] := 16#7A02;
   // UNICODE_TO_GBK[23967] := 16#EFFC;
   // UNICODE_TO_GBK[23968] := 16#7A03;
   // UNICODE_TO_GBK[23969] := 16#EFFB;
   // UNICODE_TO_GBK[23970] := 16#7A04;
   // UNICODE_TO_GBK[23971] := 16#B68F;
   // UNICODE_TO_GBK[23972] := 16#7A05;
   // UNICODE_TO_GBK[23973] := 16#B690;
   // UNICODE_TO_GBK[23974] := 16#7A06;
   // UNICODE_TO_GBK[23975] := 16#EFF9;
   // UNICODE_TO_GBK[23976] := 16#7A07;
   // UNICODE_TO_GBK[23977] := 16#B691;
   // UNICODE_TO_GBK[23978] := 16#7A08;
   // UNICODE_TO_GBK[23979] := 16#B692;
   // UNICODE_TO_GBK[23980] := 16#7A09;
   // UNICODE_TO_GBK[23981] := 16#B693;
   // UNICODE_TO_GBK[23982] := 16#7A0A;
   // UNICODE_TO_GBK[23983] := 16#B694;
   // UNICODE_TO_GBK[23984] := 16#7A0B;
   // UNICODE_TO_GBK[23985] := 16#B3CC;
   // UNICODE_TO_GBK[23986] := 16#7A0C;
   // UNICODE_TO_GBK[23987] := 16#B695;
   // UNICODE_TO_GBK[23988] := 16#7A0D;
   // UNICODE_TO_GBK[23989] := 16#C9D4;
   // UNICODE_TO_GBK[23990] := 16#7A0E;
   // UNICODE_TO_GBK[23991] := 16#CBB0;
   // UNICODE_TO_GBK[23992] := 16#7A0F;
   // UNICODE_TO_GBK[23993] := 16#B696;
   // UNICODE_TO_GBK[23994] := 16#7A10;
   // UNICODE_TO_GBK[23995] := 16#B697;
   // UNICODE_TO_GBK[23996] := 16#7A11;
   // UNICODE_TO_GBK[23997] := 16#B698;
   // UNICODE_TO_GBK[23998] := 16#7A12;
   // UNICODE_TO_GBK[23999] := 16#B699;
   // UNICODE_TO_GBK[24000] := 16#7A13;
   // UNICODE_TO_GBK[24001] := 16#B69A;
   // UNICODE_TO_GBK[24002] := 16#7A14;
   // UNICODE_TO_GBK[24003] := 16#EFFE;
   // UNICODE_TO_GBK[24004] := 16#7A15;
   // UNICODE_TO_GBK[24005] := 16#B69B;
   // UNICODE_TO_GBK[24006] := 16#7A16;
   // UNICODE_TO_GBK[24007] := 16#B69C;
   // UNICODE_TO_GBK[24008] := 16#7A17;
   // UNICODE_TO_GBK[24009] := 16#B0DE;
   // UNICODE_TO_GBK[24010] := 16#7A18;
   // UNICODE_TO_GBK[24011] := 16#B69D;
   // UNICODE_TO_GBK[24012] := 16#7A19;
   // UNICODE_TO_GBK[24013] := 16#B69E;
   // UNICODE_TO_GBK[24014] := 16#7A1A;
   // UNICODE_TO_GBK[24015] := 16#D6C9;
   // UNICODE_TO_GBK[24016] := 16#7A1B;
   // UNICODE_TO_GBK[24017] := 16#B69F;
   // UNICODE_TO_GBK[24018] := 16#7A1C;
   // UNICODE_TO_GBK[24019] := 16#B6A0;
   // UNICODE_TO_GBK[24020] := 16#7A1D;
   // UNICODE_TO_GBK[24021] := 16#B740;
   // UNICODE_TO_GBK[24022] := 16#7A1E;
   // UNICODE_TO_GBK[24023] := 16#EFFD;
   // UNICODE_TO_GBK[24024] := 16#7A1F;
   // UNICODE_TO_GBK[24025] := 16#B741;
   // UNICODE_TO_GBK[24026] := 16#7A20;
   // UNICODE_TO_GBK[24027] := 16#B3ED;
   // UNICODE_TO_GBK[24028] := 16#7A21;
   // UNICODE_TO_GBK[24029] := 16#B742;
   // UNICODE_TO_GBK[24030] := 16#7A22;
   // UNICODE_TO_GBK[24031] := 16#B743;
   // UNICODE_TO_GBK[24032] := 16#7A23;
   // UNICODE_TO_GBK[24033] := 16#F6D5;
   // UNICODE_TO_GBK[24034] := 16#7A24;
   // UNICODE_TO_GBK[24035] := 16#B744;
   // UNICODE_TO_GBK[24036] := 16#7A25;
   // UNICODE_TO_GBK[24037] := 16#B745;
   // UNICODE_TO_GBK[24038] := 16#7A26;
   // UNICODE_TO_GBK[24039] := 16#B746;
   // UNICODE_TO_GBK[24040] := 16#7A27;
   // UNICODE_TO_GBK[24041] := 16#B747;
   // UNICODE_TO_GBK[24042] := 16#7A28;
   // UNICODE_TO_GBK[24043] := 16#B748;
   // UNICODE_TO_GBK[24044] := 16#7A29;
   // UNICODE_TO_GBK[24045] := 16#B749;
   // UNICODE_TO_GBK[24046] := 16#7A2A;
   // UNICODE_TO_GBK[24047] := 16#B74A;
   // UNICODE_TO_GBK[24048] := 16#7A2B;
   // UNICODE_TO_GBK[24049] := 16#B74B;
   // UNICODE_TO_GBK[24050] := 16#7A2C;
   // UNICODE_TO_GBK[24051] := 16#B74C;
   // UNICODE_TO_GBK[24052] := 16#7A2D;
   // UNICODE_TO_GBK[24053] := 16#B74D;
   // UNICODE_TO_GBK[24054] := 16#7A2E;
   // UNICODE_TO_GBK[24055] := 16#B74E;
   // UNICODE_TO_GBK[24056] := 16#7A2F;
   // UNICODE_TO_GBK[24057] := 16#B74F;
   // UNICODE_TO_GBK[24058] := 16#7A30;
   // UNICODE_TO_GBK[24059] := 16#B750;
   // UNICODE_TO_GBK[24060] := 16#7A31;
   // UNICODE_TO_GBK[24061] := 16#B751;
   // UNICODE_TO_GBK[24062] := 16#7A32;
   // UNICODE_TO_GBK[24063] := 16#B752;
   // UNICODE_TO_GBK[24064] := 16#7A33;
   // UNICODE_TO_GBK[24065] := 16#CEC8;
   // UNICODE_TO_GBK[24066] := 16#7A34;
   // UNICODE_TO_GBK[24067] := 16#B753;
   // UNICODE_TO_GBK[24068] := 16#7A35;
   // UNICODE_TO_GBK[24069] := 16#B754;
   // UNICODE_TO_GBK[24070] := 16#7A36;
   // UNICODE_TO_GBK[24071] := 16#B755;
   // UNICODE_TO_GBK[24072] := 16#7A37;
   // UNICODE_TO_GBK[24073] := 16#F0A2;
   // UNICODE_TO_GBK[24074] := 16#7A38;
   // UNICODE_TO_GBK[24075] := 16#B756;
   // UNICODE_TO_GBK[24076] := 16#7A39;
   // UNICODE_TO_GBK[24077] := 16#F0A1;
   // UNICODE_TO_GBK[24078] := 16#7A3A;
   // UNICODE_TO_GBK[24079] := 16#B757;
   // UNICODE_TO_GBK[24080] := 16#7A3B;
   // UNICODE_TO_GBK[24081] := 16#B5BE;
   // UNICODE_TO_GBK[24082] := 16#7A3C;
   // UNICODE_TO_GBK[24083] := 16#BCDA;
   // UNICODE_TO_GBK[24084] := 16#7A3D;
   // UNICODE_TO_GBK[24085] := 16#BBFC;
   // UNICODE_TO_GBK[24086] := 16#7A3E;
   // UNICODE_TO_GBK[24087] := 16#B758;
   // UNICODE_TO_GBK[24088] := 16#7A3F;
   // UNICODE_TO_GBK[24089] := 16#B8E5;
   // UNICODE_TO_GBK[24090] := 16#7A40;
   // UNICODE_TO_GBK[24091] := 16#B759;
   // UNICODE_TO_GBK[24092] := 16#7A41;
   // UNICODE_TO_GBK[24093] := 16#B75A;
   // UNICODE_TO_GBK[24094] := 16#7A42;
   // UNICODE_TO_GBK[24095] := 16#B75B;
   // UNICODE_TO_GBK[24096] := 16#7A43;
   // UNICODE_TO_GBK[24097] := 16#B75C;
   // UNICODE_TO_GBK[24098] := 16#7A44;
   // UNICODE_TO_GBK[24099] := 16#B75D;
   // UNICODE_TO_GBK[24100] := 16#7A45;
   // UNICODE_TO_GBK[24101] := 16#B75E;
   // UNICODE_TO_GBK[24102] := 16#7A46;
   // UNICODE_TO_GBK[24103] := 16#C4C2;
   // UNICODE_TO_GBK[24104] := 16#7A47;
   // UNICODE_TO_GBK[24105] := 16#B75F;
   // UNICODE_TO_GBK[24106] := 16#7A48;
   // UNICODE_TO_GBK[24107] := 16#B760;
   // UNICODE_TO_GBK[24108] := 16#7A49;
   // UNICODE_TO_GBK[24109] := 16#B761;
   // UNICODE_TO_GBK[24110] := 16#7A4A;
   // UNICODE_TO_GBK[24111] := 16#B762;
   // UNICODE_TO_GBK[24112] := 16#7A4B;
   // UNICODE_TO_GBK[24113] := 16#B763;
   // UNICODE_TO_GBK[24114] := 16#7A4C;
   // UNICODE_TO_GBK[24115] := 16#B764;
   // UNICODE_TO_GBK[24116] := 16#7A4D;
   // UNICODE_TO_GBK[24117] := 16#B765;
   // UNICODE_TO_GBK[24118] := 16#7A4E;
   // UNICODE_TO_GBK[24119] := 16#B766;
   // UNICODE_TO_GBK[24120] := 16#7A4F;
   // UNICODE_TO_GBK[24121] := 16#B767;
   // UNICODE_TO_GBK[24122] := 16#7A50;
   // UNICODE_TO_GBK[24123] := 16#B768;
   // UNICODE_TO_GBK[24124] := 16#7A51;
   // UNICODE_TO_GBK[24125] := 16#F0A3;
   // UNICODE_TO_GBK[24126] := 16#7A52;
   // UNICODE_TO_GBK[24127] := 16#B769;
   // UNICODE_TO_GBK[24128] := 16#7A53;
   // UNICODE_TO_GBK[24129] := 16#B76A;
   // UNICODE_TO_GBK[24130] := 16#7A54;
   // UNICODE_TO_GBK[24131] := 16#B76B;
   // UNICODE_TO_GBK[24132] := 16#7A55;
   // UNICODE_TO_GBK[24133] := 16#B76C;
   // UNICODE_TO_GBK[24134] := 16#7A56;
   // UNICODE_TO_GBK[24135] := 16#B76D;
   // UNICODE_TO_GBK[24136] := 16#7A57;
   // UNICODE_TO_GBK[24137] := 16#CBEB;
   // UNICODE_TO_GBK[24138] := 16#7A58;
   // UNICODE_TO_GBK[24139] := 16#B76E;
   // UNICODE_TO_GBK[24140] := 16#7A59;
   // UNICODE_TO_GBK[24141] := 16#B76F;
   // UNICODE_TO_GBK[24142] := 16#7A5A;
   // UNICODE_TO_GBK[24143] := 16#B770;
   // UNICODE_TO_GBK[24144] := 16#7A5B;
   // UNICODE_TO_GBK[24145] := 16#B771;
   // UNICODE_TO_GBK[24146] := 16#7A5C;
   // UNICODE_TO_GBK[24147] := 16#B772;
   // UNICODE_TO_GBK[24148] := 16#7A5D;
   // UNICODE_TO_GBK[24149] := 16#B773;
   // UNICODE_TO_GBK[24150] := 16#7A5E;
   // UNICODE_TO_GBK[24151] := 16#B774;
   // UNICODE_TO_GBK[24152] := 16#7A5F;
   // UNICODE_TO_GBK[24153] := 16#B775;
   // UNICODE_TO_GBK[24154] := 16#7A60;
   // UNICODE_TO_GBK[24155] := 16#B776;
   // UNICODE_TO_GBK[24156] := 16#7A61;
   // UNICODE_TO_GBK[24157] := 16#B777;
   // UNICODE_TO_GBK[24158] := 16#7A62;
   // UNICODE_TO_GBK[24159] := 16#B778;
   // UNICODE_TO_GBK[24160] := 16#7A63;
   // UNICODE_TO_GBK[24161] := 16#B779;
   // UNICODE_TO_GBK[24162] := 16#7A64;
   // UNICODE_TO_GBK[24163] := 16#B77A;
   // UNICODE_TO_GBK[24164] := 16#7A65;
   // UNICODE_TO_GBK[24165] := 16#B77B;
   // UNICODE_TO_GBK[24166] := 16#7A66;
   // UNICODE_TO_GBK[24167] := 16#B77C;
   // UNICODE_TO_GBK[24168] := 16#7A67;
   // UNICODE_TO_GBK[24169] := 16#B77D;
   // UNICODE_TO_GBK[24170] := 16#7A68;
   // UNICODE_TO_GBK[24171] := 16#B77E;
   // UNICODE_TO_GBK[24172] := 16#7A69;
   // UNICODE_TO_GBK[24173] := 16#B780;
   // UNICODE_TO_GBK[24174] := 16#7A6A;
   // UNICODE_TO_GBK[24175] := 16#B781;
   // UNICODE_TO_GBK[24176] := 16#7A6B;
   // UNICODE_TO_GBK[24177] := 16#B782;
   // UNICODE_TO_GBK[24178] := 16#7A6C;
   // UNICODE_TO_GBK[24179] := 16#B783;
   // UNICODE_TO_GBK[24180] := 16#7A6D;
   // UNICODE_TO_GBK[24181] := 16#B784;
   // UNICODE_TO_GBK[24182] := 16#7A6E;
   // UNICODE_TO_GBK[24183] := 16#B785;
   // UNICODE_TO_GBK[24184] := 16#7A6F;
   // UNICODE_TO_GBK[24185] := 16#B786;
   // UNICODE_TO_GBK[24186] := 16#7A70;
   // UNICODE_TO_GBK[24187] := 16#F0A6;
   // UNICODE_TO_GBK[24188] := 16#7A71;
   // UNICODE_TO_GBK[24189] := 16#B787;
   // UNICODE_TO_GBK[24190] := 16#7A72;
   // UNICODE_TO_GBK[24191] := 16#B788;
   // UNICODE_TO_GBK[24192] := 16#7A73;
   // UNICODE_TO_GBK[24193] := 16#B789;
   // UNICODE_TO_GBK[24194] := 16#7A74;
   // UNICODE_TO_GBK[24195] := 16#D1A8;
   // UNICODE_TO_GBK[24196] := 16#7A75;
   // UNICODE_TO_GBK[24197] := 16#B78A;
   // UNICODE_TO_GBK[24198] := 16#7A76;
   // UNICODE_TO_GBK[24199] := 16#BEBF;
   // UNICODE_TO_GBK[24200] := 16#7A77;
   // UNICODE_TO_GBK[24201] := 16#C7EE;
   // UNICODE_TO_GBK[24202] := 16#7A78;
   // UNICODE_TO_GBK[24203] := 16#F1B6;
   // UNICODE_TO_GBK[24204] := 16#7A79;
   // UNICODE_TO_GBK[24205] := 16#F1B7;
   // UNICODE_TO_GBK[24206] := 16#7A7A;
   // UNICODE_TO_GBK[24207] := 16#BFD5;
   // UNICODE_TO_GBK[24208] := 16#7A7B;
   // UNICODE_TO_GBK[24209] := 16#B78B;
   // UNICODE_TO_GBK[24210] := 16#7A7C;
   // UNICODE_TO_GBK[24211] := 16#B78C;
   // UNICODE_TO_GBK[24212] := 16#7A7D;
   // UNICODE_TO_GBK[24213] := 16#B78D;
   // UNICODE_TO_GBK[24214] := 16#7A7E;
   // UNICODE_TO_GBK[24215] := 16#B78E;
   // UNICODE_TO_GBK[24216] := 16#7A7F;
   // UNICODE_TO_GBK[24217] := 16#B4A9;
   // UNICODE_TO_GBK[24218] := 16#7A80;
   // UNICODE_TO_GBK[24219] := 16#F1B8;
   // UNICODE_TO_GBK[24220] := 16#7A81;
   // UNICODE_TO_GBK[24221] := 16#CDBB;
   // UNICODE_TO_GBK[24222] := 16#7A82;
   // UNICODE_TO_GBK[24223] := 16#B78F;
   // UNICODE_TO_GBK[24224] := 16#7A83;
   // UNICODE_TO_GBK[24225] := 16#C7D4;
   // UNICODE_TO_GBK[24226] := 16#7A84;
   // UNICODE_TO_GBK[24227] := 16#D5AD;
   // UNICODE_TO_GBK[24228] := 16#7A85;
   // UNICODE_TO_GBK[24229] := 16#B790;
   // UNICODE_TO_GBK[24230] := 16#7A86;
   // UNICODE_TO_GBK[24231] := 16#F1B9;
   // UNICODE_TO_GBK[24232] := 16#7A87;
   // UNICODE_TO_GBK[24233] := 16#B791;
   // UNICODE_TO_GBK[24234] := 16#7A88;
   // UNICODE_TO_GBK[24235] := 16#F1BA;
   // UNICODE_TO_GBK[24236] := 16#7A89;
   // UNICODE_TO_GBK[24237] := 16#B792;
   // UNICODE_TO_GBK[24238] := 16#7A8A;
   // UNICODE_TO_GBK[24239] := 16#B793;
   // UNICODE_TO_GBK[24240] := 16#7A8B;
   // UNICODE_TO_GBK[24241] := 16#B794;
   // UNICODE_TO_GBK[24242] := 16#7A8C;
   // UNICODE_TO_GBK[24243] := 16#B795;
   // UNICODE_TO_GBK[24244] := 16#7A8D;
   // UNICODE_TO_GBK[24245] := 16#C7CF;
   // UNICODE_TO_GBK[24246] := 16#7A8E;
   // UNICODE_TO_GBK[24247] := 16#B796;
   // UNICODE_TO_GBK[24248] := 16#7A8F;
   // UNICODE_TO_GBK[24249] := 16#B797;
   // UNICODE_TO_GBK[24250] := 16#7A90;
   // UNICODE_TO_GBK[24251] := 16#B798;
   // UNICODE_TO_GBK[24252] := 16#7A91;
   // UNICODE_TO_GBK[24253] := 16#D2A4;
   // UNICODE_TO_GBK[24254] := 16#7A92;
   // UNICODE_TO_GBK[24255] := 16#D6CF;
   // UNICODE_TO_GBK[24256] := 16#7A93;
   // UNICODE_TO_GBK[24257] := 16#B799;
   // UNICODE_TO_GBK[24258] := 16#7A94;
   // UNICODE_TO_GBK[24259] := 16#B79A;
   // UNICODE_TO_GBK[24260] := 16#7A95;
   // UNICODE_TO_GBK[24261] := 16#F1BB;
   // UNICODE_TO_GBK[24262] := 16#7A96;
   // UNICODE_TO_GBK[24263] := 16#BDD1;
   // UNICODE_TO_GBK[24264] := 16#7A97;
   // UNICODE_TO_GBK[24265] := 16#B4B0;
   // UNICODE_TO_GBK[24266] := 16#7A98;
   // UNICODE_TO_GBK[24267] := 16#BEBD;
   // UNICODE_TO_GBK[24268] := 16#7A99;
   // UNICODE_TO_GBK[24269] := 16#B79B;
   // UNICODE_TO_GBK[24270] := 16#7A9A;
   // UNICODE_TO_GBK[24271] := 16#B79C;
   // UNICODE_TO_GBK[24272] := 16#7A9B;
   // UNICODE_TO_GBK[24273] := 16#B79D;
   // UNICODE_TO_GBK[24274] := 16#7A9C;
   // UNICODE_TO_GBK[24275] := 16#B4DC;
   // UNICODE_TO_GBK[24276] := 16#7A9D;
   // UNICODE_TO_GBK[24277] := 16#CED1;
   // UNICODE_TO_GBK[24278] := 16#7A9E;
   // UNICODE_TO_GBK[24279] := 16#B79E;
   // UNICODE_TO_GBK[24280] := 16#7A9F;
   // UNICODE_TO_GBK[24281] := 16#BFDF;
   // UNICODE_TO_GBK[24282] := 16#7AA0;
   // UNICODE_TO_GBK[24283] := 16#F1BD;
   // UNICODE_TO_GBK[24284] := 16#7AA1;
   // UNICODE_TO_GBK[24285] := 16#B79F;
   // UNICODE_TO_GBK[24286] := 16#7AA2;
   // UNICODE_TO_GBK[24287] := 16#B7A0;
   // UNICODE_TO_GBK[24288] := 16#7AA3;
   // UNICODE_TO_GBK[24289] := 16#B840;
   // UNICODE_TO_GBK[24290] := 16#7AA4;
   // UNICODE_TO_GBK[24291] := 16#B841;
   // UNICODE_TO_GBK[24292] := 16#7AA5;
   // UNICODE_TO_GBK[24293] := 16#BFFA;
   // UNICODE_TO_GBK[24294] := 16#7AA6;
   // UNICODE_TO_GBK[24295] := 16#F1BC;
   // UNICODE_TO_GBK[24296] := 16#7AA7;
   // UNICODE_TO_GBK[24297] := 16#B842;
   // UNICODE_TO_GBK[24298] := 16#7AA8;
   // UNICODE_TO_GBK[24299] := 16#F1BF;
   // UNICODE_TO_GBK[24300] := 16#7AA9;
   // UNICODE_TO_GBK[24301] := 16#B843;
   // UNICODE_TO_GBK[24302] := 16#7AAA;
   // UNICODE_TO_GBK[24303] := 16#B844;
   // UNICODE_TO_GBK[24304] := 16#7AAB;
   // UNICODE_TO_GBK[24305] := 16#B845;
   // UNICODE_TO_GBK[24306] := 16#7AAC;
   // UNICODE_TO_GBK[24307] := 16#F1BE;
   // UNICODE_TO_GBK[24308] := 16#7AAD;
   // UNICODE_TO_GBK[24309] := 16#F1C0;
   // UNICODE_TO_GBK[24310] := 16#7AAE;
   // UNICODE_TO_GBK[24311] := 16#B846;
   // UNICODE_TO_GBK[24312] := 16#7AAF;
   // UNICODE_TO_GBK[24313] := 16#B847;
   // UNICODE_TO_GBK[24314] := 16#7AB0;
   // UNICODE_TO_GBK[24315] := 16#B848;
   // UNICODE_TO_GBK[24316] := 16#7AB1;
   // UNICODE_TO_GBK[24317] := 16#B849;
   // UNICODE_TO_GBK[24318] := 16#7AB2;
   // UNICODE_TO_GBK[24319] := 16#B84A;
   // UNICODE_TO_GBK[24320] := 16#7AB3;
   // UNICODE_TO_GBK[24321] := 16#F1C1;
   // UNICODE_TO_GBK[24322] := 16#7AB4;
   // UNICODE_TO_GBK[24323] := 16#B84B;
   // UNICODE_TO_GBK[24324] := 16#7AB5;
   // UNICODE_TO_GBK[24325] := 16#B84C;
   // UNICODE_TO_GBK[24326] := 16#7AB6;
   // UNICODE_TO_GBK[24327] := 16#B84D;
   // UNICODE_TO_GBK[24328] := 16#7AB7;
   // UNICODE_TO_GBK[24329] := 16#B84E;
   // UNICODE_TO_GBK[24330] := 16#7AB8;
   // UNICODE_TO_GBK[24331] := 16#B84F;
   // UNICODE_TO_GBK[24332] := 16#7AB9;
   // UNICODE_TO_GBK[24333] := 16#B850;
   // UNICODE_TO_GBK[24334] := 16#7ABA;
   // UNICODE_TO_GBK[24335] := 16#B851;
   // UNICODE_TO_GBK[24336] := 16#7ABB;
   // UNICODE_TO_GBK[24337] := 16#B852;
   // UNICODE_TO_GBK[24338] := 16#7ABC;
   // UNICODE_TO_GBK[24339] := 16#B853;
   // UNICODE_TO_GBK[24340] := 16#7ABD;
   // UNICODE_TO_GBK[24341] := 16#B854;
   // UNICODE_TO_GBK[24342] := 16#7ABE;
   // UNICODE_TO_GBK[24343] := 16#B855;
   // UNICODE_TO_GBK[24344] := 16#7ABF;
   // UNICODE_TO_GBK[24345] := 16#C1FE;
   // UNICODE_TO_GBK[24346] := 16#7AC0;
   // UNICODE_TO_GBK[24347] := 16#B856;
   // UNICODE_TO_GBK[24348] := 16#7AC1;
   // UNICODE_TO_GBK[24349] := 16#B857;
   // UNICODE_TO_GBK[24350] := 16#7AC2;
   // UNICODE_TO_GBK[24351] := 16#B858;
   // UNICODE_TO_GBK[24352] := 16#7AC3;
   // UNICODE_TO_GBK[24353] := 16#B859;
   // UNICODE_TO_GBK[24354] := 16#7AC4;
   // UNICODE_TO_GBK[24355] := 16#B85A;
   // UNICODE_TO_GBK[24356] := 16#7AC5;
   // UNICODE_TO_GBK[24357] := 16#B85B;
   // UNICODE_TO_GBK[24358] := 16#7AC6;
   // UNICODE_TO_GBK[24359] := 16#B85C;
   // UNICODE_TO_GBK[24360] := 16#7AC7;
   // UNICODE_TO_GBK[24361] := 16#B85D;
   // UNICODE_TO_GBK[24362] := 16#7AC8;
   // UNICODE_TO_GBK[24363] := 16#B85E;
   // UNICODE_TO_GBK[24364] := 16#7AC9;
   // UNICODE_TO_GBK[24365] := 16#B85F;
   // UNICODE_TO_GBK[24366] := 16#7ACA;
   // UNICODE_TO_GBK[24367] := 16#B860;
   // UNICODE_TO_GBK[24368] := 16#7ACB;
   // UNICODE_TO_GBK[24369] := 16#C1A2;
   // UNICODE_TO_GBK[24370] := 16#7ACC;
   // UNICODE_TO_GBK[24371] := 16#B861;
   // UNICODE_TO_GBK[24372] := 16#7ACD;
   // UNICODE_TO_GBK[24373] := 16#B862;
   // UNICODE_TO_GBK[24374] := 16#7ACE;
   // UNICODE_TO_GBK[24375] := 16#B863;
   // UNICODE_TO_GBK[24376] := 16#7ACF;
   // UNICODE_TO_GBK[24377] := 16#B864;
   // UNICODE_TO_GBK[24378] := 16#7AD0;
   // UNICODE_TO_GBK[24379] := 16#B865;
   // UNICODE_TO_GBK[24380] := 16#7AD1;
   // UNICODE_TO_GBK[24381] := 16#B866;
   // UNICODE_TO_GBK[24382] := 16#7AD2;
   // UNICODE_TO_GBK[24383] := 16#B867;
   // UNICODE_TO_GBK[24384] := 16#7AD3;
   // UNICODE_TO_GBK[24385] := 16#B868;
   // UNICODE_TO_GBK[24386] := 16#7AD4;
   // UNICODE_TO_GBK[24387] := 16#B869;
   // UNICODE_TO_GBK[24388] := 16#7AD5;
   // UNICODE_TO_GBK[24389] := 16#B86A;
   // UNICODE_TO_GBK[24390] := 16#7AD6;
   // UNICODE_TO_GBK[24391] := 16#CAFA;
   // UNICODE_TO_GBK[24392] := 16#7AD7;
   // UNICODE_TO_GBK[24393] := 16#B86B;
   // UNICODE_TO_GBK[24394] := 16#7AD8;
   // UNICODE_TO_GBK[24395] := 16#B86C;
   // UNICODE_TO_GBK[24396] := 16#7AD9;
   // UNICODE_TO_GBK[24397] := 16#D5BE;
   // UNICODE_TO_GBK[24398] := 16#7ADA;
   // UNICODE_TO_GBK[24399] := 16#B86D;
   // UNICODE_TO_GBK[24400] := 16#7ADB;
   // UNICODE_TO_GBK[24401] := 16#B86E;
   // UNICODE_TO_GBK[24402] := 16#7ADC;
   // UNICODE_TO_GBK[24403] := 16#B86F;
   // UNICODE_TO_GBK[24404] := 16#7ADD;
   // UNICODE_TO_GBK[24405] := 16#B870;
   // UNICODE_TO_GBK[24406] := 16#7ADE;
   // UNICODE_TO_GBK[24407] := 16#BEBA;
   // UNICODE_TO_GBK[24408] := 16#7ADF;
   // UNICODE_TO_GBK[24409] := 16#BEB9;
   // UNICODE_TO_GBK[24410] := 16#7AE0;
   // UNICODE_TO_GBK[24411] := 16#D5C2;
   // UNICODE_TO_GBK[24412] := 16#7AE1;
   // UNICODE_TO_GBK[24413] := 16#B871;
   // UNICODE_TO_GBK[24414] := 16#7AE2;
   // UNICODE_TO_GBK[24415] := 16#B872;
   // UNICODE_TO_GBK[24416] := 16#7AE3;
   // UNICODE_TO_GBK[24417] := 16#BFA2;
   // UNICODE_TO_GBK[24418] := 16#7AE4;
   // UNICODE_TO_GBK[24419] := 16#B873;
   // UNICODE_TO_GBK[24420] := 16#7AE5;
   // UNICODE_TO_GBK[24421] := 16#CDAF;
   // UNICODE_TO_GBK[24422] := 16#7AE6;
   // UNICODE_TO_GBK[24423] := 16#F1B5;
   // UNICODE_TO_GBK[24424] := 16#7AE7;
   // UNICODE_TO_GBK[24425] := 16#B874;
   // UNICODE_TO_GBK[24426] := 16#7AE8;
   // UNICODE_TO_GBK[24427] := 16#B875;
   // UNICODE_TO_GBK[24428] := 16#7AE9;
   // UNICODE_TO_GBK[24429] := 16#B876;
   // UNICODE_TO_GBK[24430] := 16#7AEA;
   // UNICODE_TO_GBK[24431] := 16#B877;
   // UNICODE_TO_GBK[24432] := 16#7AEB;
   // UNICODE_TO_GBK[24433] := 16#B878;
   // UNICODE_TO_GBK[24434] := 16#7AEC;
   // UNICODE_TO_GBK[24435] := 16#B879;
   // UNICODE_TO_GBK[24436] := 16#7AED;
   // UNICODE_TO_GBK[24437] := 16#BDDF;
   // UNICODE_TO_GBK[24438] := 16#7AEE;
   // UNICODE_TO_GBK[24439] := 16#B87A;
   // UNICODE_TO_GBK[24440] := 16#7AEF;
   // UNICODE_TO_GBK[24441] := 16#B6CB;
   // UNICODE_TO_GBK[24442] := 16#7AF0;
   // UNICODE_TO_GBK[24443] := 16#B87B;
   // UNICODE_TO_GBK[24444] := 16#7AF1;
   // UNICODE_TO_GBK[24445] := 16#B87C;
   // UNICODE_TO_GBK[24446] := 16#7AF2;
   // UNICODE_TO_GBK[24447] := 16#B87D;
   // UNICODE_TO_GBK[24448] := 16#7AF3;
   // UNICODE_TO_GBK[24449] := 16#B87E;
   // UNICODE_TO_GBK[24450] := 16#7AF4;
   // UNICODE_TO_GBK[24451] := 16#B880;
   // UNICODE_TO_GBK[24452] := 16#7AF5;
   // UNICODE_TO_GBK[24453] := 16#B881;
   // UNICODE_TO_GBK[24454] := 16#7AF6;
   // UNICODE_TO_GBK[24455] := 16#B882;
   // UNICODE_TO_GBK[24456] := 16#7AF7;
   // UNICODE_TO_GBK[24457] := 16#B883;
   // UNICODE_TO_GBK[24458] := 16#7AF8;
   // UNICODE_TO_GBK[24459] := 16#B884;
   // UNICODE_TO_GBK[24460] := 16#7AF9;
   // UNICODE_TO_GBK[24461] := 16#D6F1;
   // UNICODE_TO_GBK[24462] := 16#7AFA;
   // UNICODE_TO_GBK[24463] := 16#F3C3;
   // UNICODE_TO_GBK[24464] := 16#7AFB;
   // UNICODE_TO_GBK[24465] := 16#B885;
   // UNICODE_TO_GBK[24466] := 16#7AFC;
   // UNICODE_TO_GBK[24467] := 16#B886;
   // UNICODE_TO_GBK[24468] := 16#7AFD;
   // UNICODE_TO_GBK[24469] := 16#F3C4;
   // UNICODE_TO_GBK[24470] := 16#7AFE;
   // UNICODE_TO_GBK[24471] := 16#B887;
   // UNICODE_TO_GBK[24472] := 16#7AFF;
   // UNICODE_TO_GBK[24473] := 16#B8CD;
   // UNICODE_TO_GBK[24474] := 16#7B00;
   // UNICODE_TO_GBK[24475] := 16#B888;
   // UNICODE_TO_GBK[24476] := 16#7B01;
   // UNICODE_TO_GBK[24477] := 16#B889;
   // UNICODE_TO_GBK[24478] := 16#7B02;
   // UNICODE_TO_GBK[24479] := 16#B88A;
   // UNICODE_TO_GBK[24480] := 16#7B03;
   // UNICODE_TO_GBK[24481] := 16#F3C6;
   // UNICODE_TO_GBK[24482] := 16#7B04;
   // UNICODE_TO_GBK[24483] := 16#F3C7;
   // UNICODE_TO_GBK[24484] := 16#7B05;
   // UNICODE_TO_GBK[24485] := 16#B88B;
   // UNICODE_TO_GBK[24486] := 16#7B06;
   // UNICODE_TO_GBK[24487] := 16#B0CA;
   // UNICODE_TO_GBK[24488] := 16#7B07;
   // UNICODE_TO_GBK[24489] := 16#B88C;
   // UNICODE_TO_GBK[24490] := 16#7B08;
   // UNICODE_TO_GBK[24491] := 16#F3C5;
   // UNICODE_TO_GBK[24492] := 16#7B09;
   // UNICODE_TO_GBK[24493] := 16#B88D;
   // UNICODE_TO_GBK[24494] := 16#7B0A;
   // UNICODE_TO_GBK[24495] := 16#F3C9;
   // UNICODE_TO_GBK[24496] := 16#7B0B;
   // UNICODE_TO_GBK[24497] := 16#CBF1;
   // UNICODE_TO_GBK[24498] := 16#7B0C;
   // UNICODE_TO_GBK[24499] := 16#B88E;
   // UNICODE_TO_GBK[24500] := 16#7B0D;
   // UNICODE_TO_GBK[24501] := 16#B88F;
   // UNICODE_TO_GBK[24502] := 16#7B0E;
   // UNICODE_TO_GBK[24503] := 16#B890;
   // UNICODE_TO_GBK[24504] := 16#7B0F;
   // UNICODE_TO_GBK[24505] := 16#F3CB;
   // UNICODE_TO_GBK[24506] := 16#7B10;
   // UNICODE_TO_GBK[24507] := 16#B891;
   // UNICODE_TO_GBK[24508] := 16#7B11;
   // UNICODE_TO_GBK[24509] := 16#D0A6;
   // UNICODE_TO_GBK[24510] := 16#7B12;
   // UNICODE_TO_GBK[24511] := 16#B892;
   // UNICODE_TO_GBK[24512] := 16#7B13;
   // UNICODE_TO_GBK[24513] := 16#B893;
   // UNICODE_TO_GBK[24514] := 16#7B14;
   // UNICODE_TO_GBK[24515] := 16#B1CA;
   // UNICODE_TO_GBK[24516] := 16#7B15;
   // UNICODE_TO_GBK[24517] := 16#F3C8;
   // UNICODE_TO_GBK[24518] := 16#7B16;
   // UNICODE_TO_GBK[24519] := 16#B894;
   // UNICODE_TO_GBK[24520] := 16#7B17;
   // UNICODE_TO_GBK[24521] := 16#B895;
   // UNICODE_TO_GBK[24522] := 16#7B18;
   // UNICODE_TO_GBK[24523] := 16#B896;
   // UNICODE_TO_GBK[24524] := 16#7B19;
   // UNICODE_TO_GBK[24525] := 16#F3CF;
   // UNICODE_TO_GBK[24526] := 16#7B1A;
   // UNICODE_TO_GBK[24527] := 16#B897;
   // UNICODE_TO_GBK[24528] := 16#7B1B;
   // UNICODE_TO_GBK[24529] := 16#B5D1;
   // UNICODE_TO_GBK[24530] := 16#7B1C;
   // UNICODE_TO_GBK[24531] := 16#B898;
   // UNICODE_TO_GBK[24532] := 16#7B1D;
   // UNICODE_TO_GBK[24533] := 16#B899;
   // UNICODE_TO_GBK[24534] := 16#7B1E;
   // UNICODE_TO_GBK[24535] := 16#F3D7;
   // UNICODE_TO_GBK[24536] := 16#7B1F;
   // UNICODE_TO_GBK[24537] := 16#B89A;
   // UNICODE_TO_GBK[24538] := 16#7B20;
   // UNICODE_TO_GBK[24539] := 16#F3D2;
   // UNICODE_TO_GBK[24540] := 16#7B21;
   // UNICODE_TO_GBK[24541] := 16#B89B;
   // UNICODE_TO_GBK[24542] := 16#7B22;
   // UNICODE_TO_GBK[24543] := 16#B89C;
   // UNICODE_TO_GBK[24544] := 16#7B23;
   // UNICODE_TO_GBK[24545] := 16#B89D;
   // UNICODE_TO_GBK[24546] := 16#7B24;
   // UNICODE_TO_GBK[24547] := 16#F3D4;
   // UNICODE_TO_GBK[24548] := 16#7B25;
   // UNICODE_TO_GBK[24549] := 16#F3D3;
   // UNICODE_TO_GBK[24550] := 16#7B26;
   // UNICODE_TO_GBK[24551] := 16#B7FB;
   // UNICODE_TO_GBK[24552] := 16#7B27;
   // UNICODE_TO_GBK[24553] := 16#B89E;
   // UNICODE_TO_GBK[24554] := 16#7B28;
   // UNICODE_TO_GBK[24555] := 16#B1BF;
   // UNICODE_TO_GBK[24556] := 16#7B29;
   // UNICODE_TO_GBK[24557] := 16#B89F;
   // UNICODE_TO_GBK[24558] := 16#7B2A;
   // UNICODE_TO_GBK[24559] := 16#F3CE;
   // UNICODE_TO_GBK[24560] := 16#7B2B;
   // UNICODE_TO_GBK[24561] := 16#F3CA;
   // UNICODE_TO_GBK[24562] := 16#7B2C;
   // UNICODE_TO_GBK[24563] := 16#B5DA;
   // UNICODE_TO_GBK[24564] := 16#7B2D;
   // UNICODE_TO_GBK[24565] := 16#B8A0;
   // UNICODE_TO_GBK[24566] := 16#7B2E;
   // UNICODE_TO_GBK[24567] := 16#F3D0;
   // UNICODE_TO_GBK[24568] := 16#7B2F;
   // UNICODE_TO_GBK[24569] := 16#B940;
   // UNICODE_TO_GBK[24570] := 16#7B30;
   // UNICODE_TO_GBK[24571] := 16#B941;
   // UNICODE_TO_GBK[24572] := 16#7B31;
   // UNICODE_TO_GBK[24573] := 16#F3D1;
   // UNICODE_TO_GBK[24574] := 16#7B32;
   // UNICODE_TO_GBK[24575] := 16#B942;
   // UNICODE_TO_GBK[24576] := 16#7B33;
   // UNICODE_TO_GBK[24577] := 16#F3D5;
   // UNICODE_TO_GBK[24578] := 16#7B34;
   // UNICODE_TO_GBK[24579] := 16#B943;
   // UNICODE_TO_GBK[24580] := 16#7B35;
   // UNICODE_TO_GBK[24581] := 16#B944;
   // UNICODE_TO_GBK[24582] := 16#7B36;
   // UNICODE_TO_GBK[24583] := 16#B945;
   // UNICODE_TO_GBK[24584] := 16#7B37;
   // UNICODE_TO_GBK[24585] := 16#B946;
   // UNICODE_TO_GBK[24586] := 16#7B38;
   // UNICODE_TO_GBK[24587] := 16#F3CD;
   // UNICODE_TO_GBK[24588] := 16#7B39;
   // UNICODE_TO_GBK[24589] := 16#B947;
   // UNICODE_TO_GBK[24590] := 16#7B3A;
   // UNICODE_TO_GBK[24591] := 16#BCE3;
   // UNICODE_TO_GBK[24592] := 16#7B3B;
   // UNICODE_TO_GBK[24593] := 16#B948;
   // UNICODE_TO_GBK[24594] := 16#7B3C;
   // UNICODE_TO_GBK[24595] := 16#C1FD;
   // UNICODE_TO_GBK[24596] := 16#7B3D;
   // UNICODE_TO_GBK[24597] := 16#B949;
   // UNICODE_TO_GBK[24598] := 16#7B3E;
   // UNICODE_TO_GBK[24599] := 16#F3D6;
   // UNICODE_TO_GBK[24600] := 16#7B3F;
   // UNICODE_TO_GBK[24601] := 16#B94A;
   // UNICODE_TO_GBK[24602] := 16#7B40;
   // UNICODE_TO_GBK[24603] := 16#B94B;
   // UNICODE_TO_GBK[24604] := 16#7B41;
   // UNICODE_TO_GBK[24605] := 16#B94C;
   // UNICODE_TO_GBK[24606] := 16#7B42;
   // UNICODE_TO_GBK[24607] := 16#B94D;
   // UNICODE_TO_GBK[24608] := 16#7B43;
   // UNICODE_TO_GBK[24609] := 16#B94E;
   // UNICODE_TO_GBK[24610] := 16#7B44;
   // UNICODE_TO_GBK[24611] := 16#B94F;
   // UNICODE_TO_GBK[24612] := 16#7B45;
   // UNICODE_TO_GBK[24613] := 16#F3DA;
   // UNICODE_TO_GBK[24614] := 16#7B46;
   // UNICODE_TO_GBK[24615] := 16#B950;
   // UNICODE_TO_GBK[24616] := 16#7B47;
   // UNICODE_TO_GBK[24617] := 16#F3CC;
   // UNICODE_TO_GBK[24618] := 16#7B48;
   // UNICODE_TO_GBK[24619] := 16#B951;
   // UNICODE_TO_GBK[24620] := 16#7B49;
   // UNICODE_TO_GBK[24621] := 16#B5C8;
   // UNICODE_TO_GBK[24622] := 16#7B4A;
   // UNICODE_TO_GBK[24623] := 16#B952;
   // UNICODE_TO_GBK[24624] := 16#7B4B;
   // UNICODE_TO_GBK[24625] := 16#BDEE;
   // UNICODE_TO_GBK[24626] := 16#7B4C;
   // UNICODE_TO_GBK[24627] := 16#F3DC;
   // UNICODE_TO_GBK[24628] := 16#7B4D;
   // UNICODE_TO_GBK[24629] := 16#B953;
   // UNICODE_TO_GBK[24630] := 16#7B4E;
   // UNICODE_TO_GBK[24631] := 16#B954;
   // UNICODE_TO_GBK[24632] := 16#7B4F;
   // UNICODE_TO_GBK[24633] := 16#B7A4;
   // UNICODE_TO_GBK[24634] := 16#7B50;
   // UNICODE_TO_GBK[24635] := 16#BFF0;
   // UNICODE_TO_GBK[24636] := 16#7B51;
   // UNICODE_TO_GBK[24637] := 16#D6FE;
   // UNICODE_TO_GBK[24638] := 16#7B52;
   // UNICODE_TO_GBK[24639] := 16#CDB2;
   // UNICODE_TO_GBK[24640] := 16#7B53;
   // UNICODE_TO_GBK[24641] := 16#B955;
   // UNICODE_TO_GBK[24642] := 16#7B54;
   // UNICODE_TO_GBK[24643] := 16#B4F0;
   // UNICODE_TO_GBK[24644] := 16#7B55;
   // UNICODE_TO_GBK[24645] := 16#B956;
   // UNICODE_TO_GBK[24646] := 16#7B56;
   // UNICODE_TO_GBK[24647] := 16#B2DF;
   // UNICODE_TO_GBK[24648] := 16#7B57;
   // UNICODE_TO_GBK[24649] := 16#B957;
   // UNICODE_TO_GBK[24650] := 16#7B58;
   // UNICODE_TO_GBK[24651] := 16#F3D8;
   // UNICODE_TO_GBK[24652] := 16#7B59;
   // UNICODE_TO_GBK[24653] := 16#B958;
   // UNICODE_TO_GBK[24654] := 16#7B5A;
   // UNICODE_TO_GBK[24655] := 16#F3D9;
   // UNICODE_TO_GBK[24656] := 16#7B5B;
   // UNICODE_TO_GBK[24657] := 16#C9B8;
   // UNICODE_TO_GBK[24658] := 16#7B5C;
   // UNICODE_TO_GBK[24659] := 16#B959;
   // UNICODE_TO_GBK[24660] := 16#7B5D;
   // UNICODE_TO_GBK[24661] := 16#F3DD;
   // UNICODE_TO_GBK[24662] := 16#7B5E;
   // UNICODE_TO_GBK[24663] := 16#B95A;
   // UNICODE_TO_GBK[24664] := 16#7B5F;
   // UNICODE_TO_GBK[24665] := 16#B95B;
   // UNICODE_TO_GBK[24666] := 16#7B60;
   // UNICODE_TO_GBK[24667] := 16#F3DE;
   // UNICODE_TO_GBK[24668] := 16#7B61;
   // UNICODE_TO_GBK[24669] := 16#B95C;
   // UNICODE_TO_GBK[24670] := 16#7B62;
   // UNICODE_TO_GBK[24671] := 16#F3E1;
   // UNICODE_TO_GBK[24672] := 16#7B63;
   // UNICODE_TO_GBK[24673] := 16#B95D;
   // UNICODE_TO_GBK[24674] := 16#7B64;
   // UNICODE_TO_GBK[24675] := 16#B95E;
   // UNICODE_TO_GBK[24676] := 16#7B65;
   // UNICODE_TO_GBK[24677] := 16#B95F;
   // UNICODE_TO_GBK[24678] := 16#7B66;
   // UNICODE_TO_GBK[24679] := 16#B960;
   // UNICODE_TO_GBK[24680] := 16#7B67;
   // UNICODE_TO_GBK[24681] := 16#B961;
   // UNICODE_TO_GBK[24682] := 16#7B68;
   // UNICODE_TO_GBK[24683] := 16#B962;
   // UNICODE_TO_GBK[24684] := 16#7B69;
   // UNICODE_TO_GBK[24685] := 16#B963;
   // UNICODE_TO_GBK[24686] := 16#7B6A;
   // UNICODE_TO_GBK[24687] := 16#B964;
   // UNICODE_TO_GBK[24688] := 16#7B6B;
   // UNICODE_TO_GBK[24689] := 16#B965;
   // UNICODE_TO_GBK[24690] := 16#7B6C;
   // UNICODE_TO_GBK[24691] := 16#B966;
   // UNICODE_TO_GBK[24692] := 16#7B6D;
   // UNICODE_TO_GBK[24693] := 16#B967;
   // UNICODE_TO_GBK[24694] := 16#7B6E;
   // UNICODE_TO_GBK[24695] := 16#F3DF;
   // UNICODE_TO_GBK[24696] := 16#7B6F;
   // UNICODE_TO_GBK[24697] := 16#B968;
   // UNICODE_TO_GBK[24698] := 16#7B70;
   // UNICODE_TO_GBK[24699] := 16#B969;
   // UNICODE_TO_GBK[24700] := 16#7B71;
   // UNICODE_TO_GBK[24701] := 16#F3E3;
   // UNICODE_TO_GBK[24702] := 16#7B72;
   // UNICODE_TO_GBK[24703] := 16#F3E2;
   // UNICODE_TO_GBK[24704] := 16#7B73;
   // UNICODE_TO_GBK[24705] := 16#B96A;
   // UNICODE_TO_GBK[24706] := 16#7B74;
   // UNICODE_TO_GBK[24707] := 16#B96B;
   // UNICODE_TO_GBK[24708] := 16#7B75;
   // UNICODE_TO_GBK[24709] := 16#F3DB;
   // UNICODE_TO_GBK[24710] := 16#7B76;
   // UNICODE_TO_GBK[24711] := 16#B96C;
   // UNICODE_TO_GBK[24712] := 16#7B77;
   // UNICODE_TO_GBK[24713] := 16#BFEA;
   // UNICODE_TO_GBK[24714] := 16#7B78;
   // UNICODE_TO_GBK[24715] := 16#B96D;
   // UNICODE_TO_GBK[24716] := 16#7B79;
   // UNICODE_TO_GBK[24717] := 16#B3EF;
   // UNICODE_TO_GBK[24718] := 16#7B7A;
   // UNICODE_TO_GBK[24719] := 16#B96E;
   // UNICODE_TO_GBK[24720] := 16#7B7B;
   // UNICODE_TO_GBK[24721] := 16#F3E0;
   // UNICODE_TO_GBK[24722] := 16#7B7C;
   // UNICODE_TO_GBK[24723] := 16#B96F;
   // UNICODE_TO_GBK[24724] := 16#7B7D;
   // UNICODE_TO_GBK[24725] := 16#B970;
   // UNICODE_TO_GBK[24726] := 16#7B7E;
   // UNICODE_TO_GBK[24727] := 16#C7A9;
   // UNICODE_TO_GBK[24728] := 16#7B7F;
   // UNICODE_TO_GBK[24729] := 16#B971;
   // UNICODE_TO_GBK[24730] := 16#7B80;
   // UNICODE_TO_GBK[24731] := 16#BCF2;
   // UNICODE_TO_GBK[24732] := 16#7B81;
   // UNICODE_TO_GBK[24733] := 16#B972;
   // UNICODE_TO_GBK[24734] := 16#7B82;
   // UNICODE_TO_GBK[24735] := 16#B973;
   // UNICODE_TO_GBK[24736] := 16#7B83;
   // UNICODE_TO_GBK[24737] := 16#B974;
   // UNICODE_TO_GBK[24738] := 16#7B84;
   // UNICODE_TO_GBK[24739] := 16#B975;
   // UNICODE_TO_GBK[24740] := 16#7B85;
   // UNICODE_TO_GBK[24741] := 16#F3EB;
   // UNICODE_TO_GBK[24742] := 16#7B86;
   // UNICODE_TO_GBK[24743] := 16#B976;
   // UNICODE_TO_GBK[24744] := 16#7B87;
   // UNICODE_TO_GBK[24745] := 16#B977;
   // UNICODE_TO_GBK[24746] := 16#7B88;
   // UNICODE_TO_GBK[24747] := 16#B978;
   // UNICODE_TO_GBK[24748] := 16#7B89;
   // UNICODE_TO_GBK[24749] := 16#B979;
   // UNICODE_TO_GBK[24750] := 16#7B8A;
   // UNICODE_TO_GBK[24751] := 16#B97A;
   // UNICODE_TO_GBK[24752] := 16#7B8B;
   // UNICODE_TO_GBK[24753] := 16#B97B;
   // UNICODE_TO_GBK[24754] := 16#7B8C;
   // UNICODE_TO_GBK[24755] := 16#B97C;
   // UNICODE_TO_GBK[24756] := 16#7B8D;
   // UNICODE_TO_GBK[24757] := 16#B9BF;
   // UNICODE_TO_GBK[24758] := 16#7B8E;
   // UNICODE_TO_GBK[24759] := 16#B97D;
   // UNICODE_TO_GBK[24760] := 16#7B8F;
   // UNICODE_TO_GBK[24761] := 16#B97E;
   // UNICODE_TO_GBK[24762] := 16#7B90;
   // UNICODE_TO_GBK[24763] := 16#F3E4;
   // UNICODE_TO_GBK[24764] := 16#7B91;
   // UNICODE_TO_GBK[24765] := 16#B980;
   // UNICODE_TO_GBK[24766] := 16#7B92;
   // UNICODE_TO_GBK[24767] := 16#B981;
   // UNICODE_TO_GBK[24768] := 16#7B93;
   // UNICODE_TO_GBK[24769] := 16#B982;
   // UNICODE_TO_GBK[24770] := 16#7B94;
   // UNICODE_TO_GBK[24771] := 16#B2AD;
   // UNICODE_TO_GBK[24772] := 16#7B95;
   // UNICODE_TO_GBK[24773] := 16#BBFE;
   // UNICODE_TO_GBK[24774] := 16#7B96;
   // UNICODE_TO_GBK[24775] := 16#B983;
   // UNICODE_TO_GBK[24776] := 16#7B97;
   // UNICODE_TO_GBK[24777] := 16#CBE3;
   // UNICODE_TO_GBK[24778] := 16#7B98;
   // UNICODE_TO_GBK[24779] := 16#B984;
   // UNICODE_TO_GBK[24780] := 16#7B99;
   // UNICODE_TO_GBK[24781] := 16#B985;
   // UNICODE_TO_GBK[24782] := 16#7B9A;
   // UNICODE_TO_GBK[24783] := 16#B986;
   // UNICODE_TO_GBK[24784] := 16#7B9B;
   // UNICODE_TO_GBK[24785] := 16#B987;
   // UNICODE_TO_GBK[24786] := 16#7B9C;
   // UNICODE_TO_GBK[24787] := 16#F3ED;
   // UNICODE_TO_GBK[24788] := 16#7B9D;
   // UNICODE_TO_GBK[24789] := 16#F3E9;
   // UNICODE_TO_GBK[24790] := 16#7B9E;
   // UNICODE_TO_GBK[24791] := 16#B988;
   // UNICODE_TO_GBK[24792] := 16#7B9F;
   // UNICODE_TO_GBK[24793] := 16#B989;
   // UNICODE_TO_GBK[24794] := 16#7BA0;
   // UNICODE_TO_GBK[24795] := 16#B98A;
   // UNICODE_TO_GBK[24796] := 16#7BA1;
   // UNICODE_TO_GBK[24797] := 16#B9DC;
   // UNICODE_TO_GBK[24798] := 16#7BA2;
   // UNICODE_TO_GBK[24799] := 16#F3EE;
   // UNICODE_TO_GBK[24800] := 16#7BA3;
   // UNICODE_TO_GBK[24801] := 16#B98B;
   // UNICODE_TO_GBK[24802] := 16#7BA4;
   // UNICODE_TO_GBK[24803] := 16#B98C;
   // UNICODE_TO_GBK[24804] := 16#7BA5;
   // UNICODE_TO_GBK[24805] := 16#B98D;
   // UNICODE_TO_GBK[24806] := 16#7BA6;
   // UNICODE_TO_GBK[24807] := 16#F3E5;
   // UNICODE_TO_GBK[24808] := 16#7BA7;
   // UNICODE_TO_GBK[24809] := 16#F3E6;
   // UNICODE_TO_GBK[24810] := 16#7BA8;
   // UNICODE_TO_GBK[24811] := 16#F3EA;
   // UNICODE_TO_GBK[24812] := 16#7BA9;
   // UNICODE_TO_GBK[24813] := 16#C2E1;
   // UNICODE_TO_GBK[24814] := 16#7BAA;
   // UNICODE_TO_GBK[24815] := 16#F3EC;
   // UNICODE_TO_GBK[24816] := 16#7BAB;
   // UNICODE_TO_GBK[24817] := 16#F3EF;
   // UNICODE_TO_GBK[24818] := 16#7BAC;
   // UNICODE_TO_GBK[24819] := 16#F3E8;
   // UNICODE_TO_GBK[24820] := 16#7BAD;
   // UNICODE_TO_GBK[24821] := 16#BCFD;
   // UNICODE_TO_GBK[24822] := 16#7BAE;
   // UNICODE_TO_GBK[24823] := 16#B98E;
   // UNICODE_TO_GBK[24824] := 16#7BAF;
   // UNICODE_TO_GBK[24825] := 16#B98F;
